LIN {X 0,Y 390.091,Z 385.39,A -85,B 0,C 180,E1 -11570.909,E2 -11570.909} C_VEL
LIN {X 0,Y 390.086,Z 385.387,A -85,B 0,C 180,E1 -11574.794,E2 -11574.794} C_VEL
LIN {X 0,Y 390.035,Z 385.403,A -85,B 0,C 180,E1 -11578.497,E2 -11578.497} C_VEL
LIN {X 0,Y 390.137,Z 385.63,A -85,B 0,C 180,E1 -11579.709,E2 -11579.709} C_VEL
LIN {X 0,Y 392.088,Z 395.547,A -85,B 0,C 180,E1 -11582.802,E2 -11582.802} C_VEL
LIN {X 0,Y 392.818,Z 399.954,A -85,B 0,C 180,E1 -11584.065,E2 -11584.065} C_VEL
LIN {X 0,Y 392.519,Z 405.952,A -85,B 0,C 180,E1 -11585.682,E2 -11585.682} C_VEL
LIN {X 0,Y 391.656,Z 416.045,A -85,B 0,C 180,E1 -11588.417,E2 -11588.417} C_VEL
LIN {X 0,Y 391.304,Z 419.949,A -85,B 0,C 180,E1 -11589.465,E2 -11589.465} C_VEL
LIN {X 0,Y 392.02,Z 423.777,A -85,B 0,C 180,E1 -11589.635,E2 -11589.635} C_VEL
LIN {X 0,Y 396.828,Z 450.131,A -85,B 0,C 180,E1 -11590.386,E2 -11590.386} C_VEL
LIN {X 0,Y 395.873,Z 524.91,A -85,B 0,C 180,E1 -11591.767,E2 -11591.767} C_VEL
LIN {X 0,Y 395.475,Z 534.822,A -85,B 0,C 180,E1 -11592.049,E2 -11592.049} C_VEL
LIN {X 0,Y 394.937,Z 544.807,A -85,B 0,C 180,E1 -11592.458,E2 -11592.458} C_VEL
LIN {X 0,Y 394.337,Z 555.164,A -85,B 0,C 180,E1 -11593.032,E2 -11593.032} C_VEL
LIN {X 0,Y 393.611,Z 564.308,A -85,B 0,C 180,E1 -11593.668,E2 -11593.668} C_VEL
LIN {X 0,Y 392.873,Z 573.31,A -85,B 0,C 180,E1 -11594.436,E2 -11594.436} C_VEL
LIN {X 0,Y 392.161,Z 582.039,A -85,B 0,C 180,E1 -11595.337,E2 -11595.337} C_VEL
LIN {X 0,Y 391.493,Z 589.792,A -85,B 0,C 180,E1 -11596.287,E2 -11596.287} C_VEL
LIN {X 0,Y 390.771,Z 598.261,A -85,B 0,C 180,E1 -11597.537,E2 -11597.537} C_VEL
LIN {X 0,Y 390.161,Z 604.25,A -85,B 0,C 180,E1 -11598.572,E2 -11598.572} C_VEL
LIN {X 0,Y 389.663,Z 610.562,A -85,B 0,C 180,E1 -11599.872,E2 -11599.872} C_VEL
LIN {X 0,Y 389.257,Z 615.836,A -85,B 0,C 180,E1 -11601.173,E2 -11601.173} C_VEL
LIN {X 0,Y 388.939,Z 620.93,A -85,B 0,C 180,E1 -11602.734,E2 -11602.734} C_VEL
LIN {X 0,Y 388.733,Z 624.78,A -85,B 0,C 180,E1 -11604.24,E2 -11604.24} C_VEL
LIN {X 0,Y 388.701,Z 627.827,A -85,B 0,C 180,E1 -11605.853,E2 -11605.853} C_VEL
LIN {X 0,Y 388.635,Z 629.324,A -85,B 0,C 180,E1 -11606.89,E2 -11606.89} C_VEL
LIN {X 0,Y 388.704,Z 630.847,A -85,B 0,C 180,E1 -11608.964,E2 -11608.964} C_VEL
LIN {X 0,Y 388.708,Z 631.126,A -85,B 0,C 180,E1 -11610,E2 -11610} C_VEL
LIN {X 0,Y 388.662,Z 630.251,A -85,B 0,C 180,E1 -11612.073,E2 -11612.073} C_VEL
LIN {X 0,Y 388.635,Z 629.324,A -85,B 0,C 180,E1 -11613.11,E2 -11613.11} C_VEL
LIN {X 0,Y 388.743,Z 625.981,A -85,B 0,C 180,E1 -11615.187,E2 -11615.187} C_VEL
LIN {X 0,Y 388.846,Z 622.355,A -85,B 0,C 180,E1 -11616.747,E2 -11616.747} C_VEL
LIN {X 0,Y 389.134,Z 617.624,A -85,B 0,C 180,E1 -11618.308,E2 -11618.308} C_VEL
LIN {X 0,Y 389.573,Z 611.652,A -85,B 0,C 180,E1 -11619.868,E2 -11619.868} C_VEL
LIN {X 0,Y 390.041,Z 605.559,A -85,B 0,C 180,E1 -11621.169,E2 -11621.169} C_VEL
LIN {X 0,Y 390.61,Z 599.818,A -85,B 0,C 180,E1 -11622.205,E2 -11622.205} C_VEL
LIN {X 0,Y 391.249,Z 593.161,A -85,B 0,C 180,E1 -11623.24,E2 -11623.24} C_VEL
LIN {X 0,Y 391.95,Z 585.084,A -85,B 0,C 180,E1 -11624.303,E2 -11624.303} C_VEL
LIN {X 0,Y 392.647,Z 576.194,A -85,B 0,C 180,E1 -11625.282,E2 -11625.282} C_VEL
LIN {X 0,Y 393.374,Z 567.482,A -85,B 0,C 180,E1 -11626.077,E2 -11626.077} C_VEL
LIN {X 0,Y 394.028,Z 559.091,A -85,B 0,C 180,E1 -11626.715,E2 -11626.715} C_VEL
LIN {X 0,Y 394.748,Z 548.583,A -85,B 0,C 180,E1 -11627.35,E2 -11627.35} C_VEL
LIN {X 0,Y 395.299,Z 538.249,A -85,B 0,C 180,E1 -11627.826,E2 -11627.826} C_VEL
LIN {X 0,Y 395.794,Z 527.528,A -85,B 0,C 180,E1 -11628.171,E2 -11628.171} C_VEL
LIN {X 0,Y 396.219,Z 504.75,A -85,B 0,C 180,E1 -11628.619,E2 -11628.619} C_VEL
LIN {X 0,Y 396.764,Z 449.751,A -85,B 0,C 180,E1 -11629.624,E2 -11629.624} C_VEL
LIN {X 0,Y 391.752,Z 422.313,A -85,B 0,C 180,E1 -11630.407,E2 -11630.407} C_VEL
LIN {X 0,Y 391.326,Z 419.943,A -85,B 0,C 180,E1 -11630.534,E2 -11630.534} C_VEL
LIN {X 0,Y 392.555,Z 406.144,A -85,B 0,C 180,E1 -11634.316,E2 -11634.316} C_VEL
LIN {X 0,Y 392.878,Z 400.185,A -85,B 0,C 180,E1 -11635.942,E2 -11635.942} C_VEL
LIN {X 0,Y 391.209,Z 390.975,A -85,B 0,C 180,E1 -11638.627,E2 -11638.627} C_VEL
LIN {X 0,Y 390.107,Z 385.497,A -85,B 0,C 180,E1 -11640.369,E2 -11640.369} C_VEL
LIN {X 0,Y 390.071,Z 385.399,A -85,B 0,C 180,E1 -11644.024,E2 -11644.024} C_VEL
LIN {X 0,Y 390.048,Z 385.397,A -85,B 0,C 180,E1 -11647.551,E2 -11647.551} C_VEL
LIN {X 0,Y 390.058,Z 385.376,A -85,B 0,C 180,E1 -11650.821,E2 -11650.821} C_VEL
LIN {X 0,Y 390.061,Z 385.4,A -85,B 0,C 180,E1 -11653.886,E2 -11653.886} C_VEL
LIN {X 0,Y 390.119,Z 385.387,A -85,B 0,C 180,E1 -11656.798,E2 -11656.798} C_VEL
LIN {X 0,Y 390.079,Z 385.389,A -85,B 0,C 180,E1 -11659.563,E2 -11659.563} C_VEL
LIN {X 0,Y 390.048,Z 385.398,A -85,B 0,C 180,E1 -11662.448,E2 -11662.448} C_VEL
LIN {X 0,Y 390.068,Z 385.382,A -85,B 0,C 180,E1 -11666.045,E2 -11666.045} C_VEL
LIN {X 0,Y 390.048,Z 385.397,A -85,B 0,C 180,E1 -11668.497,E2 -11668.497} C_VEL
LIN {X 0,Y 390.117,Z 385.375,A -85,B 0,C 180,E1 -11672.069,E2 -11672.069} C_VEL
LIN {X 0,Y 390.08,Z 385.387,A -85,B 0,C 180,E1 -11675.519,E2 -11675.519} C_VEL
LIN {X 0,Y 390.055,Z 385.39,A -85,B 0,C 180,E1 -11678.877,E2 -11678.877} C_VEL
LIN {X 0,Y 390.128,Z 385.368,A -85,B 0,C 180,E1 -11682.166,E2 -11682.166} C_VEL
LIN {X 0,Y 390.146,Z 385.383,A -85,B 0,C 180,E1 -11685.392,E2 -11685.392} C_VEL
LIN {X 0,Y 390.146,Z 385.372,A -85,B 0,C 180,E1 -11688.571,E2 -11688.571} C_VEL
LIN {X 0,Y 390.343,Z 385.344,A -85,B 0,C 180,E1 -11691.993,E2 -11691.993} C_VEL
LIN {X 0,Y 390.225,Z 385.373,A -85,B 0,C 180,E1 -11694.833,E2 -11694.833} C_VEL
LIN {X 0,Y 390.418,Z 385.342,A -85,B 0,C 180,E1 -11697.936,E2 -11697.936} C_VEL
LIN {X 0,Y 390.546,Z 385.309,A -85,B 0,C 180,E1 -11699.999,E2 -11699.999} C_VEL
LIN {X 0,Y 390.314,Z 385.356,A -85,B 0,C 180,E1 -11703.096,E2 -11703.096} C_VEL
LIN {X 0,Y 390.307,Z 385.361,A -85,B 0,C 180,E1 -11706.65,E2 -11706.65} C_VEL
LIN {X 0,Y 390.204,Z 385.358,A -85,B 0,C 180,E1 -11709.328,E2 -11709.328} C_VEL
LIN {X 0,Y 390.175,Z 385.374,A -85,B 0,C 180,E1 -11712.482,E2 -11712.482} C_VEL
LIN {X 0,Y 390.137,Z 385.387,A -85,B 0,C 180,E1 -11715.676,E2 -11715.676} C_VEL
LIN {X 0,Y 390.102,Z 385.371,A -85,B 0,C 180,E1 -11718.922,E2 -11718.922} C_VEL
LIN {X 0,Y 390.036,Z 385.397,A -85,B 0,C 180,E1 -11722.234,E2 -11722.234} C_VEL
LIN {X 0,Y 390.116,Z 385.38,A -85,B 0,C 180,E1 -11725.743,E2 -11725.743} C_VEL
LIN {X 0,Y 390.054,Z 385.388,A -85,B 0,C 180,E1 -11729.109,E2 -11729.109} C_VEL
LIN {X 0,Y 390.039,Z 385.397,A -85,B 0,C 180,E1 -11732.721,E2 -11732.721} C_VEL
LIN {X 0,Y 390.053,Z 385.393,A -85,B 0,C 180,E1 -11735.825,E2 -11735.825} C_VEL
LIN {X 0,Y 390.068,Z 385.394,A -85,B 0,C 180,E1 -11739.218,E2 -11739.218} C_VEL
LIN {X 0,Y 390.041,Z 385.396,A -85,B 0,C 180,E1 -11742.374,E2 -11742.374} C_VEL
LIN {X 0,Y 390.042,Z 385.388,A -85,B 0,C 180,E1 -11745.354,E2 -11745.354} C_VEL
LIN {X 0,Y 390.046,Z 385.361,A -85,B 0,C 180,E1 -11748.189,E2 -11748.189} C_VEL
LIN {X 0,Y 390.091,Z 385.388,A -85,B 0,C 180,E1 -11750.908,E2 -11750.908} C_VEL
LIN {X 0,Y 390.082,Z 385.374,A -85,B 0,C 180,E1 -11754.793,E2 -11754.793} C_VEL
LIN {X 0,Y 390.024,Z 385.402,A -85,B 0,C 180,E1 -11758.496,E2 -11758.496} C_VEL
LIN {X 0,Y 390.113,Z 385.389,A -85,B 0,C 180,E1 -11762.07,E2 -11762.07} C_VEL
LIN {X 0,Y 390.077,Z 385.397,A -85,B 0,C 180,E1 -11765.519,E2 -11765.519} C_VEL
LIN {X 0,Y 390.052,Z 385.401,A -85,B 0,C 180,E1 -11768.878,E2 -11768.878} C_VEL
LIN {X 0,Y 390.125,Z 385.391,A -85,B 0,C 180,E1 -11772.166,E2 -11772.166} C_VEL
LIN {X 0,Y 390.14,Z 385.39,A -85,B 0,C 180,E1 -11775.392,E2 -11775.392} C_VEL
LIN {X 0,Y 390.145,Z 385.389,A -85,B 0,C 180,E1 -11778.571,E2 -11778.571} C_VEL
LIN {X 0,Y 390.382,Z 385.657,A -85,B 0,C 180,E1 -11781.829,E2 -11781.829} C_VEL
LIN {X 0,Y 390.714,Z 386.9,A -85,B 0,C 180,E1 -11782.458,E2 -11782.458} C_VEL
LIN {X 0,Y 392.085,Z 389.234,A -85,B 0,C 180,E1 -11783.567,E2 -11783.567} C_VEL
LIN {X 0,Y 394.112,Z 390.919,A -85,B 0,C 180,E1 -11785.397,E2 -11785.397} C_VEL
LIN {X 0,Y 395.582,Z 391.492,A -85,B 0,C 180,E1 -11787.454,E2 -11787.454} C_VEL
LIN {X 0,Y 396.128,Z 391.931,A -85,B 0,C 180,E1 -11788.983,E2 -11788.983} C_VEL
LIN {X 0,Y 396.323,Z 391.849,A -85,B 0,C 180,E1 -11790,E2 -11790} C_VEL
LIN {X 0,Y 396.07,Z 391.804,A -85,B 0,C 180,E1 -11791.525,E2 -11791.525} C_VEL
LIN {X 0,Y 395.354,Z 391.371,A -85,B 0,C 180,E1 -11793.057,E2 -11793.057} C_VEL
LIN {X 0,Y 393.694,Z 390.658,A -85,B 0,C 180,E1 -11794.992,E2 -11794.992} C_VEL
LIN {X 0,Y 391.898,Z 389.022,A -85,B 0,C 180,E1 -11796.564,E2 -11796.564} C_VEL
LIN {X 0,Y 390.579,Z 386.504,A -85,B 0,C 180,E1 -11797.684,E2 -11797.684} C_VEL
LIN {X 0,Y 390.34,Z 385.593,A -85,B 0,C 180,E1 -11798.281,E2 -11798.281} C_VEL
LIN {X 0,Y 390.144,Z 385.389,A -85,B 0,C 180,E1 -11801.428,E2 -11801.428} C_VEL
LIN {X 0,Y 390.139,Z 385.39,A -85,B 0,C 180,E1 -11804.607,E2 -11804.607} C_VEL
LIN {X 0,Y 390.123,Z 385.391,A -85,B 0,C 180,E1 -11807.833,E2 -11807.833} C_VEL
LIN {X 0,Y 390.051,Z 385.402,A -85,B 0,C 180,E1 -11811.122,E2 -11811.122} C_VEL
LIN {X 0,Y 390.075,Z 385.397,A -85,B 0,C 180,E1 -11814.48,E2 -11814.48} C_VEL
LIN {X 0,Y 390.11,Z 385.387,A -85,B 0,C 180,E1 -11818.025,E2 -11818.025} C_VEL
LIN {X 0,Y 390.01,Z 385.395,A -85,B 0,C 180,E1 -11820.813,E2 -11820.813} C_VEL
LIN {X 0,Y 389.336,Z 385.488,A -85,B 0,C 180,E1 -11821.675,E2 -11821.675} C_VEL
LIN {X 0,Y 386.487,Z 385.833,A -85,B 0,C 180,E1 -11823.076,E2 -11823.076} C_VEL
LIN {X 0,Y 384.087,Z 386.121,A -85,B 0,C 180,E1 -11824.209,E2 -11824.209} C_VEL
LIN {X 0,Y 383.07,Z 386.246,A -85,B 0,C 180,E1 -11825.085,E2 -11825.085} C_VEL
LIN {X 0,Y 382.993,Z 386.257,A -85,B 0,C 180,E1 -11825.381,E2 -11825.381} C_VEL
LIN {X 0,Y 383.006,Z 386.277,A -85,B 0,C 180,E1 -11828.599,E2 -11828.599} C_VEL
LIN {X 0,Y 382.997,Z 386.241,A -85,B 0,C 180,E1 -11831.345,E2 -11831.345} C_VEL
LIN {X 0,Y 382.99,Z 386.262,A -85,B 0,C 180,E1 -11834.303,E2 -11834.303} C_VEL
LIN {X 0,Y 383.032,Z 386.27,A -85,B 0,C 180,E1 -11837.244,E2 -11837.244} C_VEL
LIN {X 0,Y 383.014,Z 386.267,A -85,B 0,C 180,E1 -11840.412,E2 -11840.412} C_VEL
LIN {X 0,Y 383.019,Z 386.271,A -85,B 0,C 180,E1 -11844.045,E2 -11844.045} C_VEL
LIN {X 0,Y 382.982,Z 386.275,A -85,B 0,C 180,E1 -11847.578,E2 -11847.578} C_VEL
LIN {X 0,Y 382.999,Z 386.275,A -85,B 0,C 180,E1 -11850.302,E2 -11850.302} C_VEL
LIN {X 0,Y 383.05,Z 386.253,A -85,B 0,C 180,E1 -11852.698,E2 -11852.698} C_VEL
LIN {X 0,Y 383.045,Z 386.269,A -85,B 0,C 180,E1 -11855.04,E2 -11855.04} C_VEL
LIN {X 0,Y 382.986,Z 386.271,A -85,B 0,C 180,E1 -11858.469,E2 -11858.469} C_VEL
LIN {X 0,Y 383.056,Z 386.25,A -85,B 0,C 180,E1 -11861.827,E2 -11861.827} C_VEL
LIN {X 0,Y 383.105,Z 386.262,A -85,B 0,C 180,E1 -11865.119,E2 -11865.119} C_VEL
LIN {X 0,Y 383.1,Z 386.247,A -85,B 0,C 180,E1 -11868.359,E2 -11868.359} C_VEL
LIN {X 0,Y 383.298,Z 386.225,A -85,B 0,C 180,E1 -11871.933,E2 -11871.933} C_VEL
LIN {X 0,Y 383.194,Z 386.252,A -85,B 0,C 180,E1 -11874.739,E2 -11874.739} C_VEL
LIN {X 0,Y 383.382,Z 386.215,A -85,B 0,C 180,E1 -11877.899,E2 -11877.899} C_VEL
LIN {X 0,Y 383.513,Z 386.184,A -85,B 0,C 180,E1 -11880.001,E2 -11880.001} C_VEL
LIN {X 0,Y 383.247,Z 386.242,A -85,B 0,C 180,E1 -11883.154,E2 -11883.154} C_VEL
LIN {X 0,Y 383.282,Z 386.236,A -85,B 0,C 180,E1 -11886.317,E2 -11886.317} C_VEL
LIN {X 0,Y 383.255,Z 386.219,A -85,B 0,C 180,E1 -11888.436,E2 -11888.436} C_VEL
LIN {X 0,Y 383.092,Z 386.252,A -85,B 0,C 180,E1 -11891.643,E2 -11891.643} C_VEL
LIN {X 0,Y 383.108,Z 386.258,A -85,B 0,C 180,E1 -11894.882,E2 -11894.882} C_VEL
LIN {X 0,Y 383.059,Z 386.246,A -85,B 0,C 180,E1 -11898.174,E2 -11898.174} C_VEL
LIN {X 0,Y 382.989,Z 386.271,A -85,B 0,C 180,E1 -11901.532,E2 -11901.532} C_VEL
LIN {X 0,Y 383.048,Z 386.259,A -85,B 0,C 180,E1 -11904.961,E2 -11904.961} C_VEL
LIN {X 0,Y 383.046,Z 386.264,A -85,B 0,C 180,E1 -11908.493,E2 -11908.493} C_VEL
LIN {X 0,Y 383.034,Z 386.267,A -85,B 0,C 180,E1 -11912.148,E2 -11912.148} C_VEL
LIN {X 0,Y 383.024,Z 386.27,A -85,B 0,C 180,E1 -11915.956,E2 -11915.956} C_VEL
LIN {X 0,Y 383.02,Z 386.266,A -85,B 0,C 180,E1 -11919.589,E2 -11919.589} C_VEL
LIN {X 0,Y 383.064,Z 386.266,A -85,B 0,C 180,E1 -11922.789,E2 -11922.789} C_VEL
LIN {X 0,Y 383.006,Z 386.276,A -85,B 0,C 180,E1 -11925.792,E2 -11925.792} C_VEL
LIN {X 0,Y 382.987,Z 386.259,A -85,B 0,C 180,E1 -11928.797,E2 -11928.797} C_VEL
LIN {X 0,Y 383.001,Z 386.278,A -85,B 0,C 180,E1 -11932.097,E2 -11932.097} C_VEL
LIN {X 0,Y 383.019,Z 386.273,A -85,B 0,C 180,E1 -11935.333,E2 -11935.333} C_VEL
LIN {X 0,Y 383.054,Z 386.367,A -85,B 0,C 180,E1 -11939.308,E2 -11939.308} C_VEL
LIN {X 0,Y 384.856,Z 395.359,A -85,B 0,C 180,E1 -11942.247,E2 -11942.247} C_VEL
LIN {X 0,Y 385.877,Z 401.628,A -85,B 0,C 180,E1 -11944.081,E2 -11944.081} C_VEL
LIN {X 0,Y 385.418,Z 408.77,A -85,B 0,C 180,E1 -11946.032,E2 -11946.032} C_VEL
LIN {X 0,Y 384.406,Z 419.746,A -85,B 0,C 180,E1 -11949.079,E2 -11949.079} C_VEL
LIN {X 0,Y 384.957,Z 422.907,A -85,B 0,C 180,E1 -11949.232,E2 -11949.232} C_VEL
LIN {X 0,Y 390.121,Z 450.943,A -85,B 0,C 180,E1 -11950.054,E2 -11950.054} C_VEL
LIN {X 0,Y 389.125,Z 524.715,A -85,B 0,C 180,E1 -11951.439,E2 -11951.439} C_VEL
LIN {X 0,Y 388.735,Z 534.627,A -85,B 0,C 180,E1 -11951.727,E2 -11951.727} C_VEL
LIN {X 0,Y 388.167,Z 544.612,A -85,B 0,C 180,E1 -11952.142,E2 -11952.142} C_VEL
LIN {X 0,Y 387.54,Z 554.969,A -85,B 0,C 180,E1 -11952.725,E2 -11952.725} C_VEL
LIN {X 0,Y 386.787,Z 564.113,A -85,B 0,C 180,E1 -11953.371,E2 -11953.371} C_VEL
LIN {X 0,Y 386.009,Z 573.115,A -85,B 0,C 180,E1 -11954.152,E2 -11954.152} C_VEL
LIN {X 0,Y 385.274,Z 581.844,A -85,B 0,C 180,E1 -11955.069,E2 -11955.069} C_VEL
LIN {X 0,Y 384.554,Z 589.767,A -85,B 0,C 180,E1 -11956.06,E2 -11956.06} C_VEL
LIN {X 0,Y 383.821,Z 598.065,A -85,B 0,C 180,E1 -11957.307,E2 -11957.307} C_VEL
LIN {X 0,Y 383.177,Z 604.054,A -85,B 0,C 180,E1 -11958.361,E2 -11958.361} C_VEL
LIN {X 0,Y 382.659,Z 610.367,A -85,B 0,C 180,E1 -11959.685,E2 -11959.685} C_VEL
LIN {X 0,Y 382.213,Z 615.64,A -85,B 0,C 180,E1 -11961.009,E2 -11961.009} C_VEL
LIN {X 0,Y 381.867,Z 620.734,A -85,B 0,C 180,E1 -11962.598,E2 -11962.598} C_VEL
LIN {X 0,Y 381.69,Z 624.065,A -85,B 0,C 180,E1 -11963.88,E2 -11963.88} C_VEL
LIN {X 0,Y 381.626,Z 627.632,A -85,B 0,C 180,E1 -11965.776,E2 -11965.776} C_VEL
LIN {X 0,Y 381.546,Z 629.129,A -85,B 0,C 180,E1 -11966.833,E2 -11966.833} C_VEL
LIN {X 0,Y 381.603,Z 630.652,A -85,B 0,C 180,E1 -11968.945,E2 -11968.945} C_VEL
LIN {X 0,Y 381.622,Z 630.932,A -85,B 0,C 180,E1 -11970,E2 -11970} C_VEL
LIN {X 0,Y 381.56,Z 630.056,A -85,B 0,C 180,E1 -11972.111,E2 -11972.111} C_VEL
LIN {X 0,Y 381.547,Z 629.129,A -85,B 0,C 180,E1 -11973.168,E2 -11973.168} C_VEL
LIN {X 0,Y 381.643,Z 625.785,A -85,B 0,C 180,E1 -11975.283,E2 -11975.283} C_VEL
LIN {X 0,Y 381.782,Z 622.16,A -85,B 0,C 180,E1 -11976.872,E2 -11976.872} C_VEL
LIN {X 0,Y 382.067,Z 617.428,A -85,B 0,C 180,E1 -11978.462,E2 -11978.462} C_VEL
LIN {X 0,Y 382.535,Z 611.456,A -85,B 0,C 180,E1 -11980.052,E2 -11980.052} C_VEL
LIN {X 0,Y 383.054,Z 605.363,A -85,B 0,C 180,E1 -11981.375,E2 -11981.375} C_VEL
LIN {X 0,Y 383.634,Z 599.622,A -85,B 0,C 180,E1 -11982.431,E2 -11982.431} C_VEL
LIN {X 0,Y 384.306,Z 592.965,A -85,B 0,C 180,E1 -11983.484,E2 -11983.484} C_VEL
LIN {X 0,Y 385.037,Z 584.888,A -85,B 0,C 180,E1 -11984.566,E2 -11984.566} C_VEL
LIN {X 0,Y 385.701,Z 577.049,A -85,B 0,C 180,E1 -11985.455,E2 -11985.455} C_VEL
LIN {X 0,Y 386.559,Z 567.287,A -85,B 0,C 180,E1 -11986.368,E2 -11986.368} C_VEL
LIN {X 0,Y 387.249,Z 558.896,A -85,B 0,C 180,E1 -11987.016,E2 -11987.016} C_VEL
LIN {X 0,Y 387.973,Z 548.388,A -85,B 0,C 180,E1 -11987.663,E2 -11987.663} C_VEL
LIN {X 0,Y 388.546,Z 538.054,A -85,B 0,C 180,E1 -11988.147,E2 -11988.147} C_VEL
LIN {X 0,Y 389.058,Z 527.333,A -85,B 0,C 180,E1 -11988.497,E2 -11988.497} C_VEL
LIN {X 0,Y 389.484,Z 504.554,A -85,B 0,C 180,E1 -11988.953,E2 -11988.953} C_VEL
LIN {X 0,Y 390.081,Z 450.645,A -85,B 0,C 180,E1 -11989.953,E2 -11989.953} C_VEL
LIN {X 0,Y 385.105,Z 423.546,A -85,B 0,C 180,E1 -11990.747,E2 -11990.747} C_VEL
LIN {X 0,Y 384.434,Z 420.018,A -85,B 0,C 180,E1 -11990.885,E2 -11990.885} C_VEL
LIN {X 0,Y 384.538,Z 417.771,A -85,B 0,C 180,E1 -11991.44,E2 -11991.44} C_VEL
LIN {X 0,Y 385.789,Z 404.956,A -85,B 0,C 180,E1 -11995.059,E2 -11995.059} C_VEL
LIN {X 0,Y 385.771,Z 400.514,A -85,B 0,C 180,E1 -11996.315,E2 -11996.315} C_VEL
LIN {X 0,Y 384.047,Z 391.334,A -85,B 0,C 180,E1 -11999.056,E2 -11999.056} C_VEL
LIN {X 0,Y 383.056,Z 386.368,A -85,B 0,C 180,E1 -12000.692,E2 -12000.692} C_VEL
LIN {X 0,Y 383.021,Z 386.273,A -85,B 0,C 180,E1 -12004.667,E2 -12004.667} C_VEL
LIN {X 0,Y 383.004,Z 386.278,A -85,B 0,C 180,E1 -12007.904,E2 -12007.904} C_VEL
LIN {X 0,Y 382.985,Z 386.259,A -85,B 0,C 180,E1 -12011.347,E2 -12011.347} C_VEL
LIN {X 0,Y 383.009,Z 386.274,A -85,B 0,C 180,E1 -12014.305,E2 -12014.305} C_VEL
LIN {X 0,Y 383.077,Z 386.265,A -85,B 0,C 180,E1 -12017.249,E2 -12017.249} C_VEL
LIN {X 0,Y 383.023,Z 386.265,A -85,B 0,C 180,E1 -12020.412,E2 -12020.412} C_VEL
LIN {X 0,Y 383.027,Z 386.269,A -85,B 0,C 180,E1 -12024.044,E2 -12024.044} C_VEL
LIN {X 0,Y 383.037,Z 386.267,A -85,B 0,C 180,E1 -12027.852,E2 -12027.852} C_VEL
LIN {X 0,Y 383.064,Z 386.258,A -85,B 0,C 180,E1 -12031.72,E2 -12031.72} C_VEL
LIN {X 0,Y 383.052,Z 386.259,A -85,B 0,C 180,E1 -12035.039,E2 -12035.039} C_VEL
LIN {X 0,Y 382.993,Z 386.271,A -85,B 0,C 180,E1 -12038.468,E2 -12038.468} C_VEL
LIN {X 0,Y 383.063,Z 386.245,A -85,B 0,C 180,E1 -12041.826,E2 -12041.826} C_VEL
LIN {X 0,Y 383.112,Z 386.257,A -85,B 0,C 180,E1 -12045.118,E2 -12045.118} C_VEL
LIN {X 0,Y 383.096,Z 386.251,A -85,B 0,C 180,E1 -12048.357,E2 -12048.357} C_VEL
LIN {X 0,Y 383.303,Z 386.218,A -85,B 0,C 180,E1 -12051.932,E2 -12051.932} C_VEL
LIN {X 0,Y 383.198,Z 386.249,A -85,B 0,C 180,E1 -12054.738,E2 -12054.738} C_VEL
LIN {X 0,Y 383.386,Z 386.218,A -85,B 0,C 180,E1 -12057.898,E2 -12057.898} C_VEL
LIN {X 0,Y 383.515,Z 386.184,A -85,B 0,C 180,E1 -12059.999,E2 -12059.999} C_VEL
LIN {X 0,Y 383.25,Z 386.236,A -85,B 0,C 180,E1 -12063.153,E2 -12063.153} C_VEL
LIN {X 0,Y 383.267,Z 386.237,A -85,B 0,C 180,E1 -12066.644,E2 -12066.644} C_VEL
LIN {X 0,Y 383.258,Z 386.228,A -85,B 0,C 180,E1 -12068.435,E2 -12068.435} C_VEL
LIN {X 0,Y 383.104,Z 386.247,A -85,B 0,C 180,E1 -12071.641,E2 -12071.641} C_VEL
LIN {X 0,Y 383.109,Z 386.261,A -85,B 0,C 180,E1 -12074.881,E2 -12074.881} C_VEL
LIN {X 0,Y 383.06,Z 386.25,A -85,B 0,C 180,E1 -12078.173,E2 -12078.173} C_VEL
LIN {X 0,Y 382.99,Z 386.271,A -85,B 0,C 180,E1 -12081.53,E2 -12081.53} C_VEL
LIN {X 0,Y 383.049,Z 386.269,A -85,B 0,C 180,E1 -12084.96,E2 -12084.96} C_VEL
LIN {X 0,Y 383.026,Z 386.261,A -85,B 0,C 180,E1 -12088.27,E2 -12088.27} C_VEL
LIN {X 0,Y 383.005,Z 386.273,A -85,B 0,C 180,E1 -12092.149,E2 -12092.149} C_VEL
LIN {X 0,Y 383.014,Z 386.258,A -85,B 0,C 180,E1 -12094.667,E2 -12094.667} C_VEL
LIN {X 0,Y 382.998,Z 386.277,A -85,B 0,C 180,E1 -12097.904,E2 -12097.904} C_VEL
LIN {X 0,Y 382.981,Z 386.27,A -85,B 0,C 180,E1 -12101.347,E2 -12101.347} C_VEL
LIN {X 0,Y 382.994,Z 386.274,A -85,B 0,C 180,E1 -12104.303,E2 -12104.303} C_VEL
LIN {X 0,Y 383.006,Z 386.24,A -85,B 0,C 180,E1 -12107.24,E2 -12107.24} C_VEL
LIN {X 0,Y 383.018,Z 386.266,A -85,B 0,C 180,E1 -12110.412,E2 -12110.412} C_VEL
LIN {X 0,Y 383.023,Z 386.262,A -85,B 0,C 180,E1 -12114.044,E2 -12114.044} C_VEL
LIN {X 0,Y 382.985,Z 386.278,A -85,B 0,C 180,E1 -12117.577,E2 -12117.577} C_VEL
LIN {X 0,Y 382.994,Z 386.262,A -85,B 0,C 180,E1 -12120.3,E2 -12120.3} C_VEL
LIN {X 0,Y 383.053,Z 386.271,A -85,B 0,C 180,E1 -12122.698,E2 -12122.698} C_VEL
LIN {X 0,Y 383.03,Z 386.274,A -85,B 0,C 180,E1 -12126.192,E2 -12126.192} C_VEL
LIN {X 0,Y 383.052,Z 386.272,A -85,B 0,C 180,E1 -12129.598,E2 -12129.598} C_VEL
LIN {X 0,Y 383.101,Z 386.267,A -85,B 0,C 180,E1 -12132.931,E2 -12132.931} C_VEL
LIN {X 0,Y 383.122,Z 386.263,A -85,B 0,C 180,E1 -12136.464,E2 -12136.464} C_VEL
LIN {X 0,Y 383.154,Z 386.531,A -85,B 0,C 180,E1 -12138.527,E2 -12138.527} C_VEL
LIN {X 0,Y 383.388,Z 387.531,A -85,B 0,C 180,E1 -12138.936,E2 -12138.936} C_VEL
LIN {X 0,Y 384.443,Z 389.598,A -85,B 0,C 180,E1 -12139.533,E2 -12139.533} C_VEL
LIN {X 0,Y 386.582,Z 391.495,A -85,B 0,C 180,E1 -12140.583,E2 -12140.583} C_VEL
LIN {X 0,Y 388.921,Z 392.828,A -85,B 0,C 180,E1 -12141.895,E2 -12141.895} C_VEL
LIN {X 0,Y 390.34,Z 395.395,A -85,B 0,C 180,E1 -12142.954,E2 -12142.954} C_VEL
LIN {X 0,Y 391.932,Z 397.07,A -85,B 0,C 180,E1 -12144.211,E2 -12144.211} C_VEL
LIN {X 0,Y 393.437,Z 398.03,A -85,B 0,C 180,E1 -12145.646,E2 -12145.646} C_VEL
LIN {X 0,Y 394.715,Z 398.539,A -85,B 0,C 180,E1 -12147.448,E2 -12147.448} C_VEL
LIN {X 0,Y 395.266,Z 398.978,A -85,B 0,C 180,E1 -12148.981,E2 -12148.981} C_VEL
LIN {X 0,Y 395.458,Z 398.896,A -85,B 0,C 180,E1 -12150,E2 -12150} C_VEL
LIN {X 0,Y 395.202,Z 398.853,A -85,B 0,C 180,E1 -12151.528,E2 -12151.528} C_VEL
LIN {X 0,Y 394.244,Z 398.355,A -85,B 0,C 180,E1 -12153.368,E2 -12153.368} C_VEL
LIN {X 0,Y 392.801,Z 397.722,A -85,B 0,C 180,E1 -12155.004,E2 -12155.004} C_VEL
LIN {X 0,Y 390.787,Z 395.983,A -85,B 0,C 180,E1 -12156.713,E2 -12156.713} C_VEL
LIN {X 0,Y 389.247,Z 393.415,A -85,B 0,C 180,E1 -12157.901,E2 -12157.901} C_VEL
LIN {X 0,Y 388.31,Z 392.289,A -85,B 0,C 180,E1 -12158.456,E2 -12158.456} C_VEL
LIN {X 0,Y 385.838,Z 391.008,A -85,B 0,C 180,E1 -12159.766,E2 -12159.766} C_VEL
LIN {X 0,Y 383.934,Z 388.794,A -85,B 0,C 180,E1 -12160.747,E2 -12160.747} C_VEL
LIN {X 0,Y 383.206,Z 386.796,A -85,B 0,C 180,E1 -12161.303,E2 -12161.303} C_VEL
LIN {X 0,Y 383.114,Z 386.297,A -85,B 0,C 180,E1 -12161.909,E2 -12161.909} C_VEL
LIN {X 0,Y 383.105,Z 386.266,A -85,B 0,C 180,E1 -12164.881,E2 -12164.881} C_VEL
LIN {X 0,Y 383.084,Z 386.268,A -85,B 0,C 180,E1 -12168.172,E2 -12168.172} C_VEL
LIN {X 0,Y 382.988,Z 386.28,A -85,B 0,C 180,E1 -12171.531,E2 -12171.531} C_VEL
LIN {X 0,Y 383.047,Z 386.273,A -85,B 0,C 180,E1 -12174.96,E2 -12174.96} C_VEL
LIN {X 0,Y 383.044,Z 386.259,A -85,B 0,C 180,E1 -12178.492,E2 -12178.492} C_VEL
LIN {X 0,Y 383.006,Z 386.277,A -85,B 0,C 180,E1 -12182.149,E2 -12182.149} C_VEL
LIN {X 0,Y 382.993,Z 386.257,A -85,B 0,C 180,E1 -12185.381,E2 -12185.381} C_VEL
LIN {X 0,Y 382.353,Z 386.347,A -85,B 0,C 180,E1 -12186.259,E2 -12186.259} C_VEL
LIN {X 0,Y 379.548,Z 386.709,A -85,B 0,C 180,E1 -12187.687,E2 -12187.687} C_VEL
LIN {X 0,Y 377.143,Z 387.008,A -85,B 0,C 180,E1 -12188.842,E2 -12188.842} C_VEL
LIN {X 0,Y 376.086,Z 387.129,A -85,B 0,C 180,E1 -12189.734,E2 -12189.734} C_VEL
LIN {X 0,Y 375.987,Z 387.134,A -85,B 0,C 180,E1 -12190.036,E2 -12190.036} C_VEL
LIN {X 0,Y 375.924,Z 387.139,A -85,B 0,C 180,E1 -12193.766,E2 -12193.766} C_VEL
LIN {X 0,Y 375.948,Z 387.156,A -85,B 0,C 180,E1 -12196.807,E2 -12196.807} C_VEL
LIN {X 0,Y 375.99,Z 387.139,A -85,B 0,C 180,E1 -12200.028,E2 -12200.028} C_VEL
LIN {X 0,Y 375.958,Z 387.149,A -85,B 0,C 180,E1 -12203.495,E2 -12203.495} C_VEL
LIN {X 0,Y 375.953,Z 387.138,A -85,B 0,C 180,E1 -12205.889,E2 -12205.889} C_VEL
LIN {X 0,Y 375.967,Z 387.15,A -85,B 0,C 180,E1 -12209.688,E2 -12209.688} C_VEL
LIN {X 0,Y 375.995,Z 387.132,A -85,B 0,C 180,E1 -12212.142,E2 -12212.142} C_VEL
LIN {X 0,Y 375.999,Z 387.141,A -85,B 0,C 180,E1 -12214.539,E2 -12214.539} C_VEL
LIN {X 0,Y 375.956,Z 387.152,A -85,B 0,C 180,E1 -12218.046,E2 -12218.046} C_VEL
LIN {X 0,Y 376.002,Z 387.127,A -85,B 0,C 180,E1 -12221.474,E2 -12221.474} C_VEL
LIN {X 0,Y 376.053,Z 387.142,A -85,B 0,C 180,E1 -12224.833,E2 -12224.833} C_VEL
LIN {X 0,Y 376.052,Z 387.128,A -85,B 0,C 180,E1 -12228.137,E2 -12228.137} C_VEL
LIN {X 0,Y 376.251,Z 387.102,A -85,B 0,C 180,E1 -12231.878,E2 -12231.878} C_VEL
LIN {X 0,Y 376.166,Z 387.129,A -85,B 0,C 180,E1 -12234.64,E2 -12234.64} C_VEL
LIN {X 0,Y 376.348,Z 387.091,A -85,B 0,C 180,E1 -12237.86,E2 -12237.86} C_VEL
LIN {X 0,Y 376.483,Z 387.059,A -85,B 0,C 180,E1 -12240.001,E2 -12240.001} C_VEL
LIN {X 0,Y 376.185,Z 387.121,A -85,B 0,C 180,E1 -12243.214,E2 -12243.214} C_VEL
LIN {X 0,Y 376.241,Z 387.112,A -85,B 0,C 180,E1 -12246.436,E2 -12246.436} C_VEL
LIN {X 0,Y 376.2,Z 387.096,A -85,B 0,C 180,E1 -12248.596,E2 -12248.596} C_VEL
LIN {X 0,Y 376.044,Z 387.131,A -85,B 0,C 180,E1 -12251.864,E2 -12251.864} C_VEL
LIN {X 0,Y 376.056,Z 387.135,A -85,B 0,C 180,E1 -12255.168,E2 -12255.168} C_VEL
LIN {X 0,Y 376.005,Z 387.123,A -85,B 0,C 180,E1 -12258.528,E2 -12258.528} C_VEL
LIN {X 0,Y 375.959,Z 387.15,A -85,B 0,C 180,E1 -12261.955,E2 -12261.955} C_VEL
LIN {X 0,Y 376.003,Z 387.137,A -85,B 0,C 180,E1 -12265.462,E2 -12265.462} C_VEL
LIN {X 0,Y 375.974,Z 387.147,A -85,B 0,C 180,E1 -12269.079,E2 -12269.079} C_VEL
LIN {X 0,Y 375.953,Z 387.143,A -85,B 0,C 180,E1 -12272.829,E2 -12272.829} C_VEL
LIN {X 0,Y 375.956,Z 387.145,A -85,B 0,C 180,E1 -12275.416,E2 -12275.416} C_VEL
LIN {X 0,Y 375.975,Z 387.148,A -85,B 0,C 180,E1 -12278.272,E2 -12278.272} C_VEL
LIN {X 0,Y 375.988,Z 387.148,A -85,B 0,C 180,E1 -12281.611,E2 -12281.611} C_VEL
LIN {X 0,Y 375.968,Z 387.149,A -85,B 0,C 180,E1 -12285.263,E2 -12285.263} C_VEL
LIN {X 0,Y 375.939,Z 387.134,A -85,B 0,C 180,E1 -12289.134,E2 -12289.134} C_VEL
LIN {X 0,Y 375.966,Z 387.156,A -85,B 0,C 180,E1 -12291.913,E2 -12291.913} C_VEL
LIN {X 0,Y 375.98,Z 387.149,A -85,B 0,C 180,E1 -12295.333,E2 -12295.333} C_VEL
LIN {X 0,Y 376.013,Z 387.276,A -85,B 0,C 180,E1 -12299.036,E2 -12299.036} C_VEL
LIN {X 0,Y 377.619,Z 395.319,A -85,B 0,C 180,E1 -12301.712,E2 -12301.712} C_VEL
LIN {X 0,Y 378.864,Z 402.487,A -85,B 0,C 180,E1 -12303.861,E2 -12303.861} C_VEL
LIN {X 0,Y 378.708,Z 407.155,A -85,B 0,C 180,E1 -12305.173,E2 -12305.173} C_VEL
LIN {X 0,Y 377.486,Z 419.566,A -85,B 0,C 180,E1 -12308.679,E2 -12308.679} C_VEL
LIN {X 0,Y 378.188,Z 423.444,A -85,B 0,C 180,E1 -12308.857,E2 -12308.857} C_VEL
LIN {X 0,Y 382.792,Z 447.926,A -85,B 0,C 180,E1 -12309.601,E2 -12309.601} C_VEL
LIN {X 0,Y 383.496,Z 452.152,A -85,B 0,C 180,E1 -12309.722,E2 -12309.722} C_VEL
LIN {X 0,Y 382.399,Z 524.52,A -85,B 0,C 180,E1 -12311.1,E2 -12311.1} C_VEL
LIN {X 0,Y 382.019,Z 534.433,A -85,B 0,C 180,E1 -12311.394,E2 -12311.394} C_VEL
LIN {X 0,Y 381.425,Z 544.417,A -85,B 0,C 180,E1 -12311.816,E2 -12311.816} C_VEL
LIN {X 0,Y 380.753,Z 554.773,A -85,B 0,C 180,E1 -12312.408,E2 -12312.408} C_VEL
LIN {X 0,Y 379.994,Z 563.918,A -85,B 0,C 180,E1 -12313.065,E2 -12313.065} C_VEL
LIN {X 0,Y 379.189,Z 572.92,A -85,B 0,C 180,E1 -12313.859,E2 -12313.859} C_VEL
LIN {X 0,Y 378.381,Z 581.648,A -85,B 0,C 180,E1 -12314.791,E2 -12314.791} C_VEL
LIN {X 0,Y 377.625,Z 589.742,A -85,B 0,C 180,E1 -12315.824,E2 -12315.824} C_VEL
LIN {X 0,Y 376.881,Z 597.87,A -85,B 0,C 180,E1 -12317.07,E2 -12317.07} C_VEL
LIN {X 0,Y 376.208,Z 603.858,A -85,B 0,C 180,E1 -12318.142,E2 -12318.142} C_VEL
LIN {X 0,Y 375.648,Z 610.171,A -85,B 0,C 180,E1 -12319.49,E2 -12319.49} C_VEL
LIN {X 0,Y 375.186,Z 615.445,A -85,B 0,C 180,E1 -12320.839,E2 -12320.839} C_VEL
LIN {X 0,Y 374.8,Z 620.538,A -85,B 0,C 180,E1 -12322.458,E2 -12322.458} C_VEL
LIN {X 0,Y 374.585,Z 624.21,A -85,B 0,C 180,E1 -12323.933,E2 -12323.933} C_VEL
LIN {X 0,Y 374.53,Z 627.436,A -85,B 0,C 180,E1 -12325.696,E2 -12325.696} C_VEL
LIN {X 0,Y 374.461,Z 628.934,A -85,B 0,C 180,E1 -12326.773,E2 -12326.773} C_VEL
LIN {X 0,Y 374.503,Z 630.457,A -85,B 0,C 180,E1 -12328.925,E2 -12328.925} C_VEL
LIN {X 0,Y 374.538,Z 630.737,A -85,B 0,C 180,E1 -12330,E2 -12330} C_VEL
LIN {X 0,Y 374.459,Z 629.861,A -85,B 0,C 180,E1 -12332.151,E2 -12332.151} C_VEL
LIN {X 0,Y 374.462,Z 628.934,A -85,B 0,C 180,E1 -12333.228,E2 -12333.228} C_VEL
LIN {X 0,Y 374.552,Z 625.589,A -85,B 0,C 180,E1 -12335.384,E2 -12335.384} C_VEL
LIN {X 0,Y 374.725,Z 621.964,A -85,B 0,C 180,E1 -12337.002,E2 -12337.002} C_VEL
LIN {X 0,Y 375.018,Z 617.232,A -85,B 0,C 180,E1 -12338.623,E2 -12338.623} C_VEL
LIN {X 0,Y 375.523,Z 611.26,A -85,B 0,C 180,E1 -12340.242,E2 -12340.242} C_VEL
LIN {X 0,Y 376.046,Z 605.166,A -85,B 0,C 180,E1 -12341.59,E2 -12341.59} C_VEL
LIN {X 0,Y 376.681,Z 599.426,A -85,B 0,C 180,E1 -12342.664,E2 -12342.664} C_VEL
LIN {X 0,Y 377.355,Z 592.769,A -85,B 0,C 180,E1 -12343.737,E2 -12343.737} C_VEL
LIN {X 0,Y 378.073,Z 585.505,A -85,B 0,C 180,E1 -12344.738,E2 -12344.738} C_VEL
LIN {X 0,Y 378.851,Z 576.853,A -85,B 0,C 180,E1 -12345.742,E2 -12345.742} C_VEL
LIN {X 0,Y 379.755,Z 567.092,A -85,B 0,C 180,E1 -12346.67,E2 -12346.67} C_VEL
LIN {X 0,Y 380.471,Z 558.701,A -85,B 0,C 180,E1 -12347.329,E2 -12347.329} C_VEL
LIN {X 0,Y 381.182,Z 548.192,A -85,B 0,C 180,E1 -12347.989,E2 -12347.989} C_VEL
LIN {X 0,Y 381.816,Z 537.859,A -85,B 0,C 180,E1 -12348.478,E2 -12348.478} C_VEL
LIN {X 0,Y 382.334,Z 527.138,A -85,B 0,C 180,E1 -12348.834,E2 -12348.834} C_VEL
LIN {X 0,Y 382.764,Z 504.359,A -85,B 0,C 180,E1 -12349.299,E2 -12349.299} C_VEL
LIN {X 0,Y 383.378,Z 451.227,A -85,B 0,C 180,E1 -12350.302,E2 -12350.302} C_VEL
LIN {X 0,Y 377.949,Z 422.096,A -85,B 0,C 180,E1 -12351.184,E2 -12351.184} C_VEL
LIN {X 0,Y 377.484,Z 419.576,A -85,B 0,C 180,E1 -12351.318,E2 -12351.318} C_VEL
LIN {X 0,Y 378.713,Z 407.26,A -85,B 0,C 180,E1 -12354.829,E2 -12354.829} C_VEL
LIN {X 0,Y 378.923,Z 402.758,A -85,B 0,C 180,E1 -12356.136,E2 -12356.136} C_VEL
LIN {X 0,Y 377.708,Z 395.599,A -85,B 0,C 180,E1 -12358.292,E2 -12358.292} C_VEL
LIN {X 0,Y 376.007,Z 387.257,A -85,B 0,C 180,E1 -12360.995,E2 -12360.995} C_VEL
LIN {X 0,Y 375.983,Z 387.15,A -85,B 0,C 180,E1 -12364.667,E2 -12364.667} C_VEL
LIN {X 0,Y 375.978,Z 387.152,A -85,B 0,C 180,E1 -12368.27,E2 -12368.27} C_VEL
LIN {X 0,Y 375.936,Z 387.139,A -85,B 0,C 180,E1 -12371.6,E2 -12371.6} C_VEL
LIN {X 0,Y 375.982,Z 387.147,A -85,B 0,C 180,E1 -12375.26,E2 -12375.26} C_VEL
LIN {X 0,Y 375.991,Z 387.147,A -85,B 0,C 180,E1 -12378.389,E2 -12378.389} C_VEL
LIN {X 0,Y 375.969,Z 387.151,A -85,B 0,C 180,E1 -12381.911,E2 -12381.911} C_VEL
LIN {X 0,Y 375.981,Z 387.14,A -85,B 0,C 180,E1 -12385.332,E2 -12385.332} C_VEL
LIN {X 0,Y 375.977,Z 387.15,A -85,B 0,C 180,E1 -12388.439,E2 -12388.439} C_VEL
LIN {X 0,Y 376.002,Z 387.132,A -85,B 0,C 180,E1 -12392.141,E2 -12392.141} C_VEL
LIN {X 0,Y 376.007,Z 387.137,A -85,B 0,C 180,E1 -12394.538,E2 -12394.538} C_VEL
LIN {X 0,Y 375.963,Z 387.15,A -85,B 0,C 180,E1 -12398.045,E2 -12398.045} C_VEL
LIN {X 0,Y 376.008,Z 387.122,A -85,B 0,C 180,E1 -12401.473,E2 -12401.473} C_VEL
LIN {X 0,Y 376.06,Z 387.135,A -85,B 0,C 180,E1 -12404.832,E2 -12404.832} C_VEL
LIN {X 0,Y 376.048,Z 387.13,A -85,B 0,C 180,E1 -12408.136,E2 -12408.136} C_VEL
LIN {X 0,Y 376.256,Z 387.094,A -85,B 0,C 180,E1 -12411.877,E2 -12411.877} C_VEL
LIN {X 0,Y 376.17,Z 387.124,A -85,B 0,C 180,E1 -12414.639,E2 -12414.639} C_VEL
LIN {X 0,Y 376.352,Z 387.094,A -85,B 0,C 180,E1 -12417.859,E2 -12417.859} C_VEL
LIN {X 0,Y 376.485,Z 387.059,A -85,B 0,C 180,E1 -12419.999,E2 -12419.999} C_VEL
LIN {X 0,Y 376.188,Z 387.116,A -85,B 0,C 180,E1 -12423.212,E2 -12423.212} C_VEL
LIN {X 0,Y 376.231,Z 387.113,A -85,B 0,C 180,E1 -12426.636,E2 -12426.636} C_VEL
LIN {X 0,Y 376.203,Z 387.107,A -85,B 0,C 180,E1 -12428.594,E2 -12428.594} C_VEL
LIN {X 0,Y 376.055,Z 387.128,A -85,B 0,C 180,E1 -12431.863,E2 -12431.863} C_VEL
LIN {X 0,Y 376.057,Z 387.142,A -85,B 0,C 180,E1 -12435.167,E2 -12435.167} C_VEL
LIN {X 0,Y 376.006,Z 387.127,A -85,B 0,C 180,E1 -12438.526,E2 -12438.526} C_VEL
LIN {X 0,Y 375.96,Z 387.152,A -85,B 0,C 180,E1 -12441.954,E2 -12441.954} C_VEL
LIN {X 0,Y 376.003,Z 387.141,A -85,B 0,C 180,E1 -12445.461,E2 -12445.461} C_VEL
LIN {X 0,Y 375.957,Z 387.143,A -85,B 0,C 180,E1 -12449.079,E2 -12449.079} C_VEL
LIN {X 0,Y 375.945,Z 387.153,A -85,B 0,C 180,E1 -12452.828,E2 -12452.828} C_VEL
LIN {X 0,Y 375.954,Z 387.142,A -85,B 0,C 180,E1 -12455.415,E2 -12455.415} C_VEL
LIN {X 0,Y 375.972,Z 387.151,A -85,B 0,C 180,E1 -12458.27,E2 -12458.27} C_VEL
LIN {X 0,Y 375.931,Z 387.15,A -85,B 0,C 180,E1 -12461.6,E2 -12461.6} C_VEL
LIN {X 0,Y 375.924,Z 387.147,A -85,B 0,C 180,E1 -12465.268,E2 -12465.268} C_VEL
LIN {X 0,Y 375.972,Z 387.121,A -85,B 0,C 180,E1 -12469.137,E2 -12469.137} C_VEL
LIN {X 0,Y 375.969,Z 387.153,A -85,B 0,C 180,E1 -12471.912,E2 -12471.912} C_VEL
LIN {X 0,Y 375.976,Z 387.127,A -85,B 0,C 180,E1 -12475.332,E2 -12475.332} C_VEL
LIN {X 0,Y 375.957,Z 387.154,A -85,B 0,C 180,E1 -12478.438,E2 -12478.438} C_VEL
LIN {X 0,Y 375.999,Z 387.146,A -85,B 0,C 180,E1 -12482.142,E2 -12482.142} C_VEL
LIN {X 0,Y 376.003,Z 387.15,A -85,B 0,C 180,E1 -12484.539,E2 -12484.539} C_VEL
LIN {X 0,Y 375.96,Z 387.156,A -85,B 0,C 180,E1 -12488.045,E2 -12488.045} C_VEL
LIN {X 0,Y 376.02,Z 387.149,A -85,B 0,C 180,E1 -12491.474,E2 -12491.474} C_VEL
LIN {X 0,Y 376.055,Z 387.144,A -85,B 0,C 180,E1 -12494.832,E2 -12494.832} C_VEL
LIN {X 0,Y 376.116,Z 387.431,A -85,B 0,C 180,E1 -12496.109,E2 -12496.109} C_VEL
LIN {X 0,Y 376.404,Z 388.517,A -85,B 0,C 180,E1 -12496.466,E2 -12496.466} C_VEL
LIN {X 0,Y 377.86,Z 391.022,A -85,B 0,C 180,E1 -12497.103,E2 -12497.103} C_VEL
LIN {X 0,Y 379.85,Z 392.579,A -85,B 0,C 180,E1 -12497.864,E2 -12497.864} C_VEL
LIN {X 0,Y 381.206,Z 393.425,A -85,B 0,C 180,E1 -12498.434,E2 -12498.434} C_VEL
LIN {X 0,Y 382.76,Z 396.024,A -85,B 0,C 180,E1 -12499.152,E2 -12499.152} C_VEL
LIN {X 0,Y 385.027,Z 398.223,A -85,B 0,C 180,E1 -12500.287,E2 -12500.287} C_VEL
LIN {X 0,Y 387.591,Z 399.678,A -85,B 0,C 180,E1 -12501.659,E2 -12501.659} C_VEL
LIN {X 0,Y 389.286,Z 402.436,A -85,B 0,C 180,E1 -12502.842,E2 -12502.842} C_VEL
LIN {X 0,Y 391.041,Z 404.135,A -85,B 0,C 180,E1 -12504.198,E2 -12504.198} C_VEL
LIN {X 0,Y 392.756,Z 405.215,A -85,B 0,C 180,E1 -12505.895,E2 -12505.895} C_VEL
LIN {X 0,Y 393.915,Z 405.599,A -85,B 0,C 180,E1 -12507.579,E2 -12507.579} C_VEL
LIN {X 0,Y 394.407,Z 406.003,A -85,B 0,C 180,E1 -12508.979,E2 -12508.979} C_VEL
LIN {X 0,Y 394.593,Z 405.943,A -85,B 0,C 180,E1 -12510,E2 -12510} C_VEL
LIN {X 0,Y 394.096,Z 405.716,A -85,B 0,C 180,E1 -12512.044,E2 -12512.044} C_VEL
LIN {X 0,Y 393.066,Z 405.32,A -85,B 0,C 180,E1 -12513.724,E2 -12513.724} C_VEL
LIN {X 0,Y 391.761,Z 404.661,A -85,B 0,C 180,E1 -12515.146,E2 -12515.146} C_VEL
LIN {X 0,Y 389.867,Z 403.121,A -85,B 0,C 180,E1 -12516.729,E2 -12516.729} C_VEL
LIN {X 0,Y 388.033,Z 400.487,A -85,B 0,C 180,E1 -12518.061,E2 -12518.061} C_VEL
LIN {X 0,Y 387.37,Z 399.381,A -85,B 0,C 180,E1 -12518.476,E2 -12518.476} C_VEL
LIN {X 0,Y 384.676,Z 397.976,A -85,B 0,C 180,E1 -12519.88,E2 -12519.88} C_VEL
LIN {X 0,Y 382.363,Z 395.516,A -85,B 0,C 180,E1 -12521.027,E2 -12521.027} C_VEL
LIN {X 0,Y 380.869,Z 393.117,A -85,B 0,C 180,E1 -12521.711,E2 -12521.711} C_VEL
LIN {X 0,Y 378.467,Z 391.617,A -85,B 0,C 180,E1 -12522.67,E2 -12522.67} C_VEL
LIN {X 0,Y 376.702,Z 389.286,A -85,B 0,C 180,E1 -12523.377,E2 -12523.377} C_VEL
LIN {X 0,Y 376.2,Z 387.748,A -85,B 0,C 180,E1 -12523.729,E2 -12523.729} C_VEL
LIN {X 0,Y 376.063,Z 387.166,A -85,B 0,C 180,E1 -12524.336,E2 -12524.336} C_VEL
LIN {X 0,Y 376.039,Z 387.146,A -85,B 0,C 180,E1 -12527.607,E2 -12527.607} C_VEL
LIN {X 0,Y 375.973,Z 387.155,A -85,B 0,C 180,E1 -12530.832,E2 -12530.832} C_VEL
LIN {X 0,Y 375.988,Z 387.152,A -85,B 0,C 180,E1 -12534.281,E2 -12534.281} C_VEL
LIN {X 0,Y 376.014,Z 387.15,A -85,B 0,C 180,E1 -12536.652,E2 -12536.652} C_VEL
LIN {X 0,Y 375.971,Z 387.135,A -85,B 0,C 180,E1 -12539.078,E2 -12539.078} C_VEL
LIN {X 0,Y 375.944,Z 387.148,A -85,B 0,C 180,E1 -12542.828,E2 -12542.828} C_VEL
LIN {X 0,Y 375.952,Z 387.135,A -85,B 0,C 180,E1 -12545.415,E2 -12545.415} C_VEL
LIN {X 0,Y 375.976,Z 387.153,A -85,B 0,C 180,E1 -12548.272,E2 -12548.272} C_VEL
LIN {X 0,Y 375.987,Z 387.134,A -85,B 0,C 180,E1 -12550.036,E2 -12550.036} C_VEL
LIN {X 0,Y 375.269,Z 387.207,A -85,B 0,C 180,E1 -12550.93,E2 -12550.93} C_VEL
LIN {X 0,Y 372.358,Z 387.563,A -85,B 0,C 180,E1 -12552.381,E2 -12552.381} C_VEL
LIN {X 0,Y 369.946,Z 387.877,A -85,B 0,C 180,E1 -12553.555,E2 -12553.555} C_VEL
LIN {X 0,Y 368.955,Z 388.011,A -85,B 0,C 180,E1 -12554.464,E2 -12554.464} C_VEL
LIN {X 0,Y 368.896,Z 388.022,A -85,B 0,C 180,E1 -12554.772,E2 -12554.772} C_VEL
LIN {X 0,Y 368.903,Z 388.028,A -85,B 0,C 180,E1 -12558.181,E2 -12558.181} C_VEL
LIN {X 0,Y 368.905,Z 388.031,A -85,B 0,C 180,E1 -12561.359,E2 -12561.359} C_VEL
LIN {X 0,Y 368.93,Z 388.012,A -85,B 0,C 180,E1 -12565.147,E2 -12565.147} C_VEL
LIN {X 0,Y 368.922,Z 388.03,A -85,B 0,C 180,E1 -12569.047,E2 -12569.047} C_VEL
LIN {X 0,Y 368.981,Z 388.009,A -85,B 0,C 180,E1 -12571.565,E2 -12571.565} C_VEL
LIN {X 0,Y 368.95,Z 388.024,A -85,B 0,C 180,E1 -12575.225,E2 -12575.225} C_VEL
LIN {X 0,Y 368.931,Z 388.016,A -85,B 0,C 180,E1 -12578.974,E2 -12578.974} C_VEL
LIN {X 0,Y 368.984,Z 388.005,A -85,B 0,C 180,E1 -12582.258,E2 -12582.258} C_VEL
LIN {X 0,Y 369.031,Z 388.018,A -85,B 0,C 180,E1 -12586.228,E2 -12586.228} C_VEL
LIN {X 0,Y 369.063,Z 387.985,A -85,B 0,C 180,E1 -12590.132,E2 -12590.132} C_VEL
LIN {X 0,Y 369.182,Z 387.987,A -85,B 0,C 180,E1 -12592.343,E2 -12592.343} C_VEL
LIN {X 0,Y 369.139,Z 388.005,A -85,B 0,C 180,E1 -12594.538,E2 -12594.538} C_VEL
LIN {X 0,Y 369.313,Z 387.967,A -85,B 0,C 180,E1 -12597.819,E2 -12597.819} C_VEL
LIN {X 0,Y 369.452,Z 387.934,A -85,B 0,C 180,E1 -12600.001,E2 -12600.001} C_VEL
LIN {X 0,Y 369.314,Z 387.971,A -85,B 0,C 180,E1 -12602.182,E2 -12602.182} C_VEL
LIN {X 0,Y 369.203,Z 387.987,A -85,B 0,C 180,E1 -12606.559,E2 -12606.559} C_VEL
LIN {X 0,Y 369.132,Z 387.974,A -85,B 0,C 180,E1 -12608.762,E2 -12608.762} C_VEL
LIN {X 0,Y 369,Z 388.01,A -85,B 0,C 180,E1 -12612.094,E2 -12612.094} C_VEL
LIN {X 0,Y 368.996,Z 388.015,A -85,B 0,C 180,E1 -12615.465,E2 -12615.465} C_VEL
LIN {X 0,Y 368.954,Z 388.001,A -85,B 0,C 180,E1 -12618.895,E2 -12618.895} C_VEL
LIN {X 0,Y 368.928,Z 388.03,A -85,B 0,C 180,E1 -12622.396,E2 -12622.396} C_VEL
LIN {X 0,Y 368.996,Z 388.003,A -85,B 0,C 180,E1 -12625.981,E2 -12625.981} C_VEL
LIN {X 0,Y 368.964,Z 388.021,A -85,B 0,C 180,E1 -12628.814,E2 -12628.814} C_VEL
LIN {X 0,Y 368.907,Z 388.025,A -85,B 0,C 180,E1 -12632.238,E2 -12632.238} C_VEL
LIN {X 0,Y 368.927,Z 388.02,A -85,B 0,C 180,E1 -12635.002,E2 -12635.002} C_VEL
LIN {X 0,Y 368.911,Z 388.025,A -85,B 0,C 180,E1 -12638.642,E2 -12638.642} C_VEL
LIN {X 0,Y 368.95,Z 388.029,A -85,B 0,C 180,E1 -12642.023,E2 -12642.023} C_VEL
LIN {X 0,Y 368.923,Z 388.027,A -85,B 0,C 180,E1 -12645.184,E2 -12645.184} C_VEL
LIN {X 0,Y 368.881,Z 388.02,A -85,B 0,C 180,E1 -12648.178,E2 -12648.178} C_VEL
LIN {X 0,Y 368.91,Z 388.03,A -85,B 0,C 180,E1 -12651.36,E2 -12651.36} C_VEL
LIN {X 0,Y 368.937,Z 388.024,A -85,B 0,C 180,E1 -12655.147,E2 -12655.147} C_VEL
LIN {X 0,Y 368.951,Z 388.212,A -85,B 0,C 180,E1 -12658.731,E2 -12658.731} C_VEL
LIN {X 0,Y 370.453,Z 395.676,A -85,B 0,C 180,E1 -12661.275,E2 -12661.275} C_VEL
LIN {X 0,Y 371.976,Z 404.39,A -85,B 0,C 180,E1 -12663.943,E2 -12663.943} C_VEL
LIN {X 0,Y 371.393,Z 411.553,A -85,B 0,C 180,E1 -12665.993,E2 -12665.993} C_VEL
LIN {X 0,Y 370.617,Z 419.437,A -85,B 0,C 180,E1 -12668.276,E2 -12668.276} C_VEL
LIN {X 0,Y 371.687,Z 425.119,A -85,B 0,C 180,E1 -12668.507,E2 -12668.507} C_VEL
LIN {X 0,Y 376.221,Z 449.345,A -85,B 0,C 180,E1 -12669.26,E2 -12669.26} C_VEL
LIN {X 0,Y 376.807,Z 454.758,A -85,B 0,C 180,E1 -12669.402,E2 -12669.402} C_VEL
LIN {X 0,Y 375.69,Z 524.325,A -85,B 0,C 180,E1 -12670.749,E2 -12670.749} C_VEL
LIN {X 0,Y 375.309,Z 534.238,A -85,B 0,C 180,E1 -12671.049,E2 -12671.049} C_VEL
LIN {X 0,Y 374.687,Z 544.222,A -85,B 0,C 180,E1 -12671.477,E2 -12671.477} C_VEL
LIN {X 0,Y 373.986,Z 554.578,A -85,B 0,C 180,E1 -12672.079,E2 -12672.079} C_VEL
LIN {X 0,Y 373.212,Z 563.723,A -85,B 0,C 180,E1 -12672.748,E2 -12672.748} C_VEL
LIN {X 0,Y 372.364,Z 572.724,A -85,B 0,C 180,E1 -12673.555,E2 -12673.555} C_VEL
LIN {X 0,Y 371.509,Z 581.452,A -85,B 0,C 180,E1 -12674.502,E2 -12674.502} C_VEL
LIN {X 0,Y 370.777,Z 589.077,A -85,B 0,C 180,E1 -12675.486,E2 -12675.486} C_VEL
LIN {X 0,Y 369.932,Z 597.674,A -85,B 0,C 180,E1 -12676.822,E2 -12676.822} C_VEL
LIN {X 0,Y 369.251,Z 603.663,A -85,B 0,C 180,E1 -12677.915,E2 -12677.915} C_VEL
LIN {X 0,Y 368.609,Z 609.974,A -85,B 0,C 180,E1 -12679.287,E2 -12679.287} C_VEL
LIN {X 0,Y 368.134,Z 615.248,A -85,B 0,C 180,E1 -12680.662,E2 -12680.662} C_VEL
LIN {X 0,Y 367.723,Z 620.342,A -85,B 0,C 180,E1 -12682.312,E2 -12682.312} C_VEL
LIN {X 0,Y 367.506,Z 624.279,A -85,B 0,C 180,E1 -12683.949,E2 -12683.949} C_VEL
LIN {X 0,Y 367.438,Z 627.241,A -85,B 0,C 180,E1 -12685.613,E2 -12685.613} C_VEL
LIN {X 0,Y 367.379,Z 628.739,A -85,B 0,C 180,E1 -12686.71,E2 -12686.71} C_VEL
LIN {X 0,Y 367.403,Z 630.262,A -85,B 0,C 180,E1 -12688.904,E2 -12688.904} C_VEL
LIN {X 0,Y 367.44,Z 630.542,A -85,B 0,C 180,E1 -12690,E2 -12690} C_VEL
LIN {X 0,Y 367.36,Z 629.666,A -85,B 0,C 180,E1 -12692.193,E2 -12692.193} C_VEL
LIN {X 0,Y 367.379,Z 628.739,A -85,B 0,C 180,E1 -12693.29,E2 -12693.29} C_VEL
LIN {X 0,Y 367.464,Z 625.394,A -85,B 0,C 180,E1 -12695.488,E2 -12695.488} C_VEL
LIN {X 0,Y 367.662,Z 621.769,A -85,B 0,C 180,E1 -12697.138,E2 -12697.138} C_VEL
LIN {X 0,Y 367.988,Z 617.037,A -85,B 0,C 180,E1 -12698.789,E2 -12698.789} C_VEL
LIN {X 0,Y 368.519,Z 611.065,A -85,B 0,C 180,E1 -12700.438,E2 -12700.438} C_VEL
LIN {X 0,Y 369.064,Z 604.971,A -85,B 0,C 180,E1 -12701.813,E2 -12701.813} C_VEL
LIN {X 0,Y 369.735,Z 599.23,A -85,B 0,C 180,E1 -12702.906,E2 -12702.906} C_VEL
LIN {X 0,Y 370.41,Z 592.572,A -85,B 0,C 180,E1 -12704,E2 -12704} C_VEL
LIN {X 0,Y 371.191,Z 584.93,A -85,B 0,C 180,E1 -12705.066,E2 -12705.066} C_VEL
LIN {X 0,Y 371.999,Z 576.658,A -85,B 0,C 180,E1 -12706.04,E2 -12706.04} C_VEL
LIN {X 0,Y 372.948,Z 566.896,A -85,B 0,C 180,E1 -12706.983,E2 -12706.983} C_VEL
LIN {X 0,Y 373.698,Z 558.506,A -85,B 0,C 180,E1 -12707.653,E2 -12707.653} C_VEL
LIN {X 0,Y 374.424,Z 547.997,A -85,B 0,C 180,E1 -12708.325,E2 -12708.325} C_VEL
LIN {X 0,Y 375.101,Z 537.664,A -85,B 0,C 180,E1 -12708.821,E2 -12708.821} C_VEL
LIN {X 0,Y 375.624,Z 526.943,A -85,B 0,C 180,E1 -12709.184,E2 -12709.184} C_VEL
LIN {X 0,Y 376.053,Z 504.164,A -85,B 0,C 180,E1 -12709.658,E2 -12709.658} C_VEL
LIN {X 0,Y 376.698,Z 451.945,A -85,B 0,C 180,E1 -12710.661,E2 -12710.661} C_VEL
LIN {X 0,Y 371.498,Z 424.01,A -85,B 0,C 180,E1 -12711.527,E2 -12711.527} C_VEL
LIN {X 0,Y 370.577,Z 419.456,A -85,B 0,C 180,E1 -12711.722,E2 -12711.722} C_VEL
LIN {X 0,Y 371.832,Z 407.432,A -85,B 0,C 180,E1 -12715.213,E2 -12715.213} C_VEL
LIN {X 0,Y 371.922,Z 403.569,A -85,B 0,C 180,E1 -12716.364,E2 -12716.364} C_VEL
LIN {X 0,Y 370.023,Z 393.216,A -85,B 0,C 180,E1 -12719.592,E2 -12719.592} C_VEL
LIN {X 0,Y 368.94,Z 388.12,A -85,B 0,C 180,E1 -12721.35,E2 -12721.35} C_VEL
LIN {X 0,Y 368.932,Z 388.023,A -85,B 0,C 180,E1 -12725.001,E2 -12725.001} C_VEL
LIN {X 0,Y 368.912,Z 388.03,A -85,B 0,C 180,E1 -12728.64,E2 -12728.64} C_VEL
LIN {X 0,Y 368.883,Z 388.021,A -85,B 0,C 180,E1 -12732.009,E2 -12732.009} C_VEL
LIN {X 0,Y 368.957,Z 388.022,A -85,B 0,C 180,E1 -12735.187,E2 -12735.187} C_VEL
LIN {X 0,Y 368.947,Z 388.027,A -85,B 0,C 180,E1 -12738.186,E2 -12738.186} C_VEL
LIN {X 0,Y 368.914,Z 388.024,A -85,B 0,C 180,E1 -12741.358,E2 -12741.358} C_VEL
LIN {X 0,Y 368.938,Z 388.018,A -85,B 0,C 180,E1 -12745.146,E2 -12745.146} C_VEL
LIN {X 0,Y 368.93,Z 388.027,A -85,B 0,C 180,E1 -12749.046,E2 -12749.046} C_VEL
LIN {X 0,Y 368.987,Z 388.013,A -85,B 0,C 180,E1 -12751.564,E2 -12751.564} C_VEL
LIN {X 0,Y 368.958,Z 388.015,A -85,B 0,C 180,E1 -12755.224,E2 -12755.224} C_VEL
LIN {X 0,Y 368.937,Z 388.021,A -85,B 0,C 180,E1 -12758.973,E2 -12758.973} C_VEL
LIN {X 0,Y 368.99,Z 387.999,A -85,B 0,C 180,E1 -12762.257,E2 -12762.257} C_VEL
LIN {X 0,Y 369.036,Z 388.013,A -85,B 0,C 180,E1 -12766.227,E2 -12766.227} C_VEL
LIN {X 0,Y 369.066,Z 387.979,A -85,B 0,C 180,E1 -12770.131,E2 -12770.131} C_VEL
LIN {X 0,Y 369.187,Z 387.983,A -85,B 0,C 180,E1 -12772.342,E2 -12772.342} C_VEL
LIN {X 0,Y 369.143,Z 388,A -85,B 0,C 180,E1 -12774.537,E2 -12774.537} C_VEL
LIN {X 0,Y 369.317,Z 387.97,A -85,B 0,C 180,E1 -12777.818,E2 -12777.818} C_VEL
LIN {X 0,Y 369.454,Z 387.934,A -85,B 0,C 180,E1 -12779.999,E2 -12779.999} C_VEL
LIN {X 0,Y 369.317,Z 387.967,A -85,B 0,C 180,E1 -12782.181,E2 -12782.181} C_VEL
LIN {X 0,Y 369.201,Z 387.99,A -85,B 0,C 180,E1 -12786.624,E2 -12786.624} C_VEL
LIN {X 0,Y 369.136,Z 387.987,A -85,B 0,C 180,E1 -12788.76,E2 -12788.76} C_VEL
LIN {X 0,Y 369.01,Z 388.009,A -85,B 0,C 180,E1 -12792.092,E2 -12792.092} C_VEL
LIN {X 0,Y 368.996,Z 388.023,A -85,B 0,C 180,E1 -12795.464,E2 -12795.464} C_VEL
LIN {X 0,Y 368.955,Z 388.003,A -85,B 0,C 180,E1 -12798.894,E2 -12798.894} C_VEL
LIN {X 0,Y 368.929,Z 388.026,A -85,B 0,C 180,E1 -12802.395,E2 -12802.395} C_VEL
LIN {X 0,Y 368.997,Z 388.008,A -85,B 0,C 180,E1 -12805.98,E2 -12805.98} C_VEL
LIN {X 0,Y 368.911,Z 388.029,A -85,B 0,C 180,E1 -12809.69,E2 -12809.69} C_VEL
LIN {X 0,Y 368.893,Z 388.029,A -85,B 0,C 180,E1 -12813.043,E2 -12813.043} C_VEL
LIN {X 0,Y 368.914,Z 388.027,A -85,B 0,C 180,E1 -12816.196,E2 -12816.196} C_VEL
LIN {X 0,Y 368.901,Z 388.034,A -85,B 0,C 180,E1 -12818.952,E2 -12818.952} C_VEL
LIN {X 0,Y 368.878,Z 388.033,A -85,B 0,C 180,E1 -12822.009,E2 -12822.009} C_VEL
LIN {X 0,Y 368.882,Z 388.025,A -85,B 0,C 180,E1 -12825.176,E2 -12825.176} C_VEL
LIN {X 0,Y 368.89,Z 387.993,A -85,B 0,C 180,E1 -12828.179,E2 -12828.179} C_VEL
LIN {X 0,Y 368.913,Z 388.031,A -85,B 0,C 180,E1 -12831.358,E2 -12831.358} C_VEL
LIN {X 0,Y 368.933,Z 388.004,A -85,B 0,C 180,E1 -12835.146,E2 -12835.146} C_VEL
LIN {X 0,Y 368.925,Z 388.026,A -85,B 0,C 180,E1 -12839.046,E2 -12839.046} C_VEL
LIN {X 0,Y 368.983,Z 388.01,A -85,B 0,C 180,E1 -12841.564,E2 -12841.564} C_VEL
LIN {X 0,Y 368.954,Z 388.029,A -85,B 0,C 180,E1 -12845.224,E2 -12845.224} C_VEL
LIN {X 0,Y 368.934,Z 388.031,A -85,B 0,C 180,E1 -12848.973,E2 -12848.973} C_VEL
LIN {X 0,Y 368.987,Z 388.025,A -85,B 0,C 180,E1 -12852.257,E2 -12852.257} C_VEL
LIN {X 0,Y 369.013,Z 388.291,A -85,B 0,C 180,E1 -12854.04,E2 -12854.04} C_VEL
LIN {X 0,Y 369.278,Z 389.281,A -85,B 0,C 180,E1 -12854.353,E2 -12854.353} C_VEL
LIN {X 0,Y 370.507,Z 391.576,A -85,B 0,C 180,E1 -12854.81,E2 -12854.81} C_VEL
LIN {X 0,Y 372.884,Z 393.484,A -85,B 0,C 180,E1 -12855.608,E2 -12855.608} C_VEL
LIN {X 0,Y 373.97,Z 394.369,A -85,B 0,C 180,E1 -12855.962,E2 -12855.962} C_VEL
LIN {X 0,Y 375.971,Z 397.483,A -85,B 0,C 180,E1 -12856.76,E2 -12856.76} C_VEL
LIN {X 0,Y 378.432,Z 399.425,A -85,B 0,C 180,E1 -12857.668,E2 -12857.668} C_VEL
LIN {X 0,Y 379.535,Z 400.186,A -85,B 0,C 180,E1 -12858.131,E2 -12858.131} C_VEL
LIN {X 0,Y 381.399,Z 402.935,A -85,B 0,C 180,E1 -12858.978,E2 -12858.978} C_VEL
LIN {X 0,Y 383.705,Z 405.063,A -85,B 0,C 180,E1 -12860.095,E2 -12860.095} C_VEL
LIN {X 0,Y 386.285,Z 406.572,A -85,B 0,C 180,E1 -12861.433,E2 -12861.433} C_VEL
LIN {X 0,Y 388.223,Z 409.439,A -85,B 0,C 180,E1 -12862.72,E2 -12862.72} C_VEL
LIN {X 0,Y 390.151,Z 411.179,A -85,B 0,C 180,E1 -12864.184,E2 -12864.184} C_VEL
LIN {X 0,Y 391.884,Z 412.239,A -85,B 0,C 180,E1 -12865.886,E2 -12865.886} C_VEL
LIN {X 0,Y 392.994,Z 412.614,A -85,B 0,C 180,E1 -12867.456,E2 -12867.456} C_VEL
LIN {X 0,Y 393.545,Z 413.05,A -85,B 0,C 180,E1 -12868.976,E2 -12868.976} C_VEL
LIN {X 0,Y 393.727,Z 412.99,A -85,B 0,C 180,E1 -12870,E2 -12870} C_VEL
LIN {X 0,Y 393.467,Z 412.924,A -85,B 0,C 180,E1 -12871.535,E2 -12871.535} C_VEL
LIN {X 0,Y 392.738,Z 412.499,A -85,B 0,C 180,E1 -12873.077,E2 -12873.077} C_VEL
LIN {X 0,Y 391.175,Z 411.894,A -85,B 0,C 180,E1 -12874.895,E2 -12874.895} C_VEL
LIN {X 0,Y 389.129,Z 410.384,A -85,B 0,C 180,E1 -12876.619,E2 -12876.619} C_VEL
LIN {X 0,Y 387.297,Z 408.114,A -85,B 0,C 180,E1 -12877.941,E2 -12877.941} C_VEL
LIN {X 0,Y 385.95,Z 406.185,A -85,B 0,C 180,E1 -12878.772,E2 -12878.772} C_VEL
LIN {X 0,Y 383.231,Z 404.738,A -85,B 0,C 180,E1 -12880.134,E2 -12880.134} C_VEL
LIN {X 0,Y 380.894,Z 402.373,A -85,B 0,C 180,E1 -12881.238,E2 -12881.238} C_VEL
LIN {X 0,Y 379.161,Z 399.793,A -85,B 0,C 180,E1 -12882.036,E2 -12882.036} C_VEL
LIN {X 0,Y 376.572,Z 398.102,A -85,B 0,C 180,E1 -12883.01,E2 -12883.01} C_VEL
LIN {X 0,Y 374.518,Z 395.358,A -85,B 0,C 180,E1 -12883.833,E2 -12883.833} C_VEL
LIN {X 0,Y 373.643,Z 393.895,A -85,B 0,C 180,E1 -12884.153,E2 -12884.153} C_VEL
LIN {X 0,Y 370.851,Z 391.975,A -85,B 0,C 180,E1 -12885.068,E2 -12885.068} C_VEL
LIN {X 0,Y 369.451,Z 389.794,A -85,B 0,C 180,E1 -12885.569,E2 -12885.569} C_VEL
LIN {X 0,Y 369.036,Z 388.426,A -85,B 0,C 180,E1 -12885.888,E2 -12885.888} C_VEL
LIN {X 0,Y 368.971,Z 388.026,A -85,B 0,C 180,E1 -12886.601,E2 -12886.601} C_VEL
LIN {X 0,Y 368.932,Z 388.031,A -85,B 0,C 180,E1 -12890.053,E2 -12890.053} C_VEL
LIN {X 0,Y 368.94,Z 388.03,A -85,B 0,C 180,E1 -12893.887,E2 -12893.887} C_VEL
LIN {X 0,Y 368.966,Z 388.027,A -85,B 0,C 180,E1 -12897.203,E2 -12897.203} C_VEL
LIN {X 0,Y 368.917,Z 388.014,A -85,B 0,C 180,E1 -12899.689,E2 -12899.689} C_VEL
LIN {X 0,Y 368.89,Z 388.018,A -85,B 0,C 180,E1 -12903.538,E2 -12903.538} C_VEL
LIN {X 0,Y 368.901,Z 388.029,A -85,B 0,C 180,E1 -12906.857,E2 -12906.857} C_VEL
LIN {X 0,Y 368.946,Z 388.003,A -85,B 0,C 180,E1 -12910.364,E2 -12910.364} C_VEL
LIN {X 0,Y 368.876,Z 388.012,A -85,B 0,C 180,E1 -12913.616,E2 -12913.616} C_VEL
LIN {X 0,Y 368.896,Z 388.022,A -85,B 0,C 180,E1 -12914.772,E2 -12914.772} C_VEL
LIN {X 0,Y 368.284,Z 388.11,A -85,B 0,C 180,E1 -12915.683,E2 -12915.683} C_VEL
LIN {X 0,Y 365.436,Z 388.464,A -85,B 0,C 180,E1 -12917.164,E2 -12917.164} C_VEL
LIN {X 0,Y 362.99,Z 388.761,A -85,B 0,C 180,E1 -12918.362,E2 -12918.362} C_VEL
LIN {X 0,Y 361.941,Z 388.886,A -85,B 0,C 180,E1 -12919.289,E2 -12919.289} C_VEL
LIN {X 0,Y 361.858,Z 388.896,A -85,B 0,C 180,E1 -12919.603,E2 -12919.603} C_VEL
LIN {X 0,Y 361.866,Z 388.908,A -85,B 0,C 180,E1 -12922.983,E2 -12922.983} C_VEL
LIN {X 0,Y 361.852,Z 388.9,A -85,B 0,C 180,E1 -12926.631,E2 -12926.631} C_VEL
LIN {X 0,Y 361.871,Z 388.906,A -85,B 0,C 180,E1 -12929.673,E2 -12929.673} C_VEL
LIN {X 0,Y 361.948,Z 388.884,A -85,B 0,C 180,E1 -12933.475,E2 -12933.475} C_VEL
LIN {X 0,Y 361.883,Z 388.904,A -85,B 0,C 180,E1 -12937.145,E2 -12937.145} C_VEL
LIN {X 0,Y 361.9,Z 388.88,A -85,B 0,C 180,E1 -12940.724,E2 -12940.724} C_VEL
LIN {X 0,Y 361.926,Z 388.896,A -85,B 0,C 180,E1 -12943.066,E2 -12943.066} C_VEL
LIN {X 0,Y 361.993,Z 388.89,A -85,B 0,C 180,E1 -12946.528,E2 -12946.528} C_VEL
LIN {X 0,Y 362.027,Z 388.86,A -85,B 0,C 180,E1 -12949.939,E2 -12949.939} C_VEL
LIN {X 0,Y 362.145,Z 388.861,A -85,B 0,C 180,E1 -12952.193,E2 -12952.193} C_VEL
LIN {X 0,Y 362.113,Z 388.881,A -85,B 0,C 180,E1 -12954.432,E2 -12954.432} C_VEL
LIN {X 0,Y 362.277,Z 388.844,A -85,B 0,C 180,E1 -12957.777,E2 -12957.777} C_VEL
LIN {X 0,Y 362.422,Z 388.809,A -85,B 0,C 180,E1 -12960.001,E2 -12960.001} C_VEL
LIN {X 0,Y 362.278,Z 388.847,A -85,B 0,C 180,E1 -12962.224,E2 -12962.224} C_VEL
LIN {X 0,Y 362.167,Z 388.862,A -85,B 0,C 180,E1 -12966.687,E2 -12966.687} C_VEL
LIN {X 0,Y 362.069,Z 388.852,A -85,B 0,C 180,E1 -12968.934,E2 -12968.934} C_VEL
LIN {X 0,Y 361.955,Z 388.891,A -85,B 0,C 180,E1 -12972.333,E2 -12972.333} C_VEL
LIN {X 0,Y 361.959,Z 388.894,A -85,B 0,C 180,E1 -12974.621,E2 -12974.621} C_VEL
LIN {X 0,Y 361.952,Z 388.872,A -85,B 0,C 180,E1 -12978.1,E2 -12978.1} C_VEL
LIN {X 0,Y 361.888,Z 388.9,A -85,B 0,C 180,E1 -12981.654,E2 -12981.654} C_VEL
LIN {X 0,Y 361.925,Z 388.89,A -85,B 0,C 180,E1 -12985.291,E2 -12985.291} C_VEL
LIN {X 0,Y 361.919,Z 388.884,A -85,B 0,C 180,E1 -12987.779,E2 -12987.779} C_VEL
LIN {X 0,Y 361.857,Z 388.91,A -85,B 0,C 180,E1 -12991.628,E2 -12991.628} C_VEL
LIN {X 0,Y 361.872,Z 388.899,A -85,B 0,C 180,E1 -12995.346,E2 -12995.346} C_VEL
LIN {X 0,Y 361.873,Z 388.9,A -85,B 0,C 180,E1 -12999.029,E2 -12999.029} C_VEL
LIN {X 0,Y 361.888,Z 388.906,A -85,B 0,C 180,E1 -13002.442,E2 -13002.442} C_VEL
LIN {X 0,Y 361.846,Z 388.911,A -85,B 0,C 180,E1 -13005.637,E2 -13005.637} C_VEL
LIN {X 0,Y 361.834,Z 388.89,A -85,B 0,C 180,E1 -13009.246,E2 -13009.246} C_VEL
LIN {X 0,Y 361.865,Z 388.906,A -85,B 0,C 180,E1 -13012.778,E2 -13012.778} C_VEL
LIN {X 0,Y 361.856,Z 388.912,A -85,B 0,C 180,E1 -13015.721,E2 -13015.721} C_VEL
LIN {X 0,Y 361.945,Z 389.069,A -85,B 0,C 180,E1 -13018.382,E2 -13018.382} C_VEL
LIN {X 0,Y 363.483,Z 396.883,A -85,B 0,C 180,E1 -13021.094,E2 -13021.094} C_VEL
LIN {X 0,Y 364.986,Z 405.25,A -85,B 0,C 180,E1 -13023.713,E2 -13023.713} C_VEL
LIN {X 0,Y 364.548,Z 411.358,A -85,B 0,C 180,E1 -13025.513,E2 -13025.513} C_VEL
LIN {X 0,Y 363.737,Z 419.229,A -85,B 0,C 180,E1 -13027.841,E2 -13027.841} C_VEL
LIN {X 0,Y 364.736,Z 424.517,A -85,B 0,C 180,E1 -13028.068,E2 -13028.068} C_VEL
LIN {X 0,Y 369.524,Z 449.828,A -85,B 0,C 180,E1 -13028.881,E2 -13028.881} C_VEL
LIN {X 0,Y 370.15,Z 455.397,A -85,B 0,C 180,E1 -13029.031,E2 -13029.031} C_VEL
LIN {X 0,Y 368.997,Z 524.13,A -85,B 0,C 180,E1 -13030.386,E2 -13030.386} C_VEL
LIN {X 0,Y 368.614,Z 534.043,A -85,B 0,C 180,E1 -13030.691,E2 -13030.691} C_VEL
LIN {X 0,Y 367.976,Z 544.027,A -85,B 0,C 180,E1 -13031.126,E2 -13031.126} C_VEL
LIN {X 0,Y 367.212,Z 554.383,A -85,B 0,C 180,E1 -13031.736,E2 -13031.736} C_VEL
LIN {X 0,Y 366.435,Z 563.528,A -85,B 0,C 180,E1 -13032.418,E2 -13032.418} C_VEL
LIN {X 0,Y 365.521,Z 572.528,A -85,B 0,C 180,E1 -13033.238,E2 -13033.238} C_VEL
LIN {X 0,Y 364.664,Z 581.257,A -85,B 0,C 180,E1 -13034.204,E2 -13034.204} C_VEL
LIN {X 0,Y 363.846,Z 589.232,A -85,B 0,C 180,E1 -13035.257,E2 -13035.257} C_VEL
LIN {X 0,Y 362.977,Z 597.478,A -85,B 0,C 180,E1 -13036.565,E2 -13036.565} C_VEL
LIN {X 0,Y 362.276,Z 603.467,A -85,B 0,C 180,E1 -13037.679,E2 -13037.679} C_VEL
LIN {X 0,Y 361.586,Z 609.778,A -85,B 0,C 180,E1 -13039.076,E2 -13039.076} C_VEL
LIN {X 0,Y 361.084,Z 615.052,A -85,B 0,C 180,E1 -13040.478,E2 -13040.478} C_VEL
LIN {X 0,Y 360.673,Z 620.146,A -85,B 0,C 180,E1 -13042.161,E2 -13042.161} C_VEL
LIN {X 0,Y 360.5,Z 622.987,A -85,B 0,C 180,E1 -13043.283,E2 -13043.283} C_VEL
LIN {X 0,Y 360.35,Z 627.046,A -85,B 0,C 180,E1 -13045.526,E2 -13045.526} C_VEL
LIN {X 0,Y 360.298,Z 628.545,A -85,B 0,C 180,E1 -13046.646,E2 -13046.646} C_VEL
LIN {X 0,Y 360.303,Z 630.067,A -85,B 0,C 180,E1 -13048.883,E2 -13048.883} C_VEL
LIN {X 0,Y 360.343,Z 630.347,A -85,B 0,C 180,E1 -13050,E2 -13050} C_VEL
LIN {X 0,Y 360.265,Z 629.471,A -85,B 0,C 180,E1 -13052.236,E2 -13052.236} C_VEL
LIN {X 0,Y 360.298,Z 628.544,A -85,B 0,C 180,E1 -13053.355,E2 -13053.355} C_VEL
LIN {X 0,Y 360.365,Z 625.198,A -85,B 0,C 180,E1 -13055.596,E2 -13055.596} C_VEL
LIN {X 0,Y 360.594,Z 621.573,A -85,B 0,C 180,E1 -13057.278,E2 -13057.278} C_VEL
LIN {X 0,Y 360.932,Z 616.841,A -85,B 0,C 180,E1 -13058.962,E2 -13058.962} C_VEL
LIN {X 0,Y 361.507,Z 610.869,A -85,B 0,C 180,E1 -13060.643,E2 -13060.643} C_VEL
LIN {X 0,Y 361.939,Z 606.086,A -85,B 0,C 180,E1 -13061.764,E2 -13061.764} C_VEL
LIN {X 0,Y 362.605,Z 600.595,A -85,B 0,C 180,E1 -13062.879,E2 -13062.879} C_VEL
LIN {X 0,Y 363.497,Z 592.376,A -85,B 0,C 180,E1 -13064.271,E2 -13064.271} C_VEL
LIN {X 0,Y 364.226,Z 585.599,A -85,B 0,C 180,E1 -13065.249,E2 -13065.249} C_VEL
LIN {X 0,Y 365.166,Z 576.462,A -85,B 0,C 180,E1 -13066.348,E2 -13066.348} C_VEL
LIN {X 0,Y 366.14,Z 566.701,A -85,B 0,C 180,E1 -13067.309,E2 -13067.309} C_VEL
LIN {X 0,Y 366.937,Z 558.311,A -85,B 0,C 180,E1 -13067.99,E2 -13067.99} C_VEL
LIN {X 0,Y 367.697,Z 547.802,A -85,B 0,C 180,E1 -13068.672,E2 -13068.672} C_VEL
LIN {X 0,Y 368.415,Z 537.47,A -85,B 0,C 180,E1 -13069.176,E2 -13069.176} C_VEL
LIN {X 0,Y 368.93,Z 526.748,A -85,B 0,C 180,E1 -13069.546,E2 -13069.546} C_VEL
LIN {X 0,Y 369.386,Z 505.76,A -85,B 0,C 180,E1 -13069.991,E2 -13069.991} C_VEL
LIN {X 0,Y 370.094,Z 453,A -85,B 0,C 180,E1 -13071.021,E2 -13071.021} C_VEL
LIN {X 0,Y 365.018,Z 425.773,A -85,B 0,C 180,E1 -13071.888,E2 -13071.888} C_VEL
LIN {X 0,Y 363.701,Z 419.535,A -85,B 0,C 180,E1 -13072.127,E2 -13072.127} C_VEL
LIN {X 0,Y 363.689,Z 418.82,A -85,B 0,C 180,E1 -13072.24,E2 -13072.24} C_VEL
LIN {X 0,Y 365.005,Z 407.397,A -85,B 0,C 180,E1 -13075.672,E2 -13075.672} C_VEL
LIN {X 0,Y 364.751,Z 403.513,A -85,B 0,C 180,E1 -13076.879,E2 -13076.879} C_VEL
LIN {X 0,Y 363.059,Z 394.503,A -85,B 0,C 180,E1 -13079.767,E2 -13079.767} C_VEL
LIN {X 0,Y 361.919,Z 388.985,A -85,B 0,C 180,E1 -13081.703,E2 -13081.703} C_VEL
LIN {X 0,Y 361.871,Z 388.897,A -85,B 0,C 180,E1 -13085.636,E2 -13085.636} C_VEL
LIN {X 0,Y 361.873,Z 388.905,A -85,B 0,C 180,E1 -13089.026,E2 -13089.026} C_VEL
LIN {X 0,Y 361.84,Z 388.91,A -85,B 0,C 180,E1 -13092.828,E2 -13092.828} C_VEL
LIN {X 0,Y 361.914,Z 388.897,A -85,B 0,C 180,E1 -13095.931,E2 -13095.931} C_VEL
LIN {X 0,Y 361.908,Z 388.9,A -85,B 0,C 180,E1 -13099.231,E2 -13099.231} C_VEL
LIN {X 0,Y 361.874,Z 388.906,A -85,B 0,C 180,E1 -13102.982,E2 -13102.982} C_VEL
LIN {X 0,Y 361.863,Z 388.896,A -85,B 0,C 180,E1 -13106.629,E2 -13106.629} C_VEL
LIN {X 0,Y 361.877,Z 388.91,A -85,B 0,C 180,E1 -13109.672,E2 -13109.672} C_VEL
LIN {X 0,Y 361.955,Z 388.876,A -85,B 0,C 180,E1 -13113.475,E2 -13113.475} C_VEL
LIN {X 0,Y 361.89,Z 388.903,A -85,B 0,C 180,E1 -13117.144,E2 -13117.144} C_VEL
LIN {X 0,Y 361.906,Z 388.881,A -85,B 0,C 180,E1 -13120.723,E2 -13120.723} C_VEL
LIN {X 0,Y 361.934,Z 388.883,A -85,B 0,C 180,E1 -13123.065,E2 -13123.065} C_VEL
LIN {X 0,Y 361.998,Z 388.888,A -85,B 0,C 180,E1 -13126.527,E2 -13126.527} C_VEL
LIN {X 0,Y 362.03,Z 388.857,A -85,B 0,C 180,E1 -13129.937,E2 -13129.937} C_VEL
LIN {X 0,Y 362.145,Z 388.856,A -85,B 0,C 180,E1 -13132.192,E2 -13132.192} C_VEL
LIN {X 0,Y 362.117,Z 388.875,A -85,B 0,C 180,E1 -13134.431,E2 -13134.431} C_VEL
LIN {X 0,Y 362.281,Z 388.847,A -85,B 0,C 180,E1 -13137.776,E2 -13137.776} C_VEL
LIN {X 0,Y 362.424,Z 388.808,A -85,B 0,C 180,E1 -13139.999,E2 -13139.999} C_VEL
LIN {X 0,Y 362.281,Z 388.843,A -85,B 0,C 180,E1 -13142.223,E2 -13142.223} C_VEL
LIN {X 0,Y 362.17,Z 388.867,A -85,B 0,C 180,E1 -13146.686,E2 -13146.686} C_VEL
LIN {X 0,Y 362.073,Z 388.863,A -85,B 0,C 180,E1 -13148.933,E2 -13148.933} C_VEL
LIN {X 0,Y 361.964,Z 388.888,A -85,B 0,C 180,E1 -13152.332,E2 -13152.332} C_VEL
LIN {X 0,Y 361.96,Z 388.895,A -85,B 0,C 180,E1 -13154.62,E2 -13154.62} C_VEL
LIN {X 0,Y 361.953,Z 388.878,A -85,B 0,C 180,E1 -13158.099,E2 -13158.099} C_VEL
LIN {X 0,Y 361.889,Z 388.9,A -85,B 0,C 180,E1 -13161.652,E2 -13161.652} C_VEL
LIN {X 0,Y 361.925,Z 388.896,A -85,B 0,C 180,E1 -13165.29,E2 -13165.29} C_VEL
LIN {X 0,Y 361.905,Z 388.885,A -85,B 0,C 180,E1 -13167.779,E2 -13167.779} C_VEL
LIN {X 0,Y 361.834,Z 388.914,A -85,B 0,C 180,E1 -13171.629,E2 -13171.629} C_VEL
LIN {X 0,Y 361.871,Z 388.894,A -85,B 0,C 180,E1 -13175.344,E2 -13175.344} C_VEL
LIN {X 0,Y 361.868,Z 388.908,A -85,B 0,C 180,E1 -13179.027,E2 -13179.027} C_VEL
LIN {X 0,Y 361.833,Z 388.911,A -85,B 0,C 180,E1 -13182.828,E2 -13182.828} C_VEL
LIN {X 0,Y 361.817,Z 388.897,A -85,B 0,C 180,E1 -13185.946,E2 -13185.946} C_VEL
LIN {X 0,Y 361.864,Z 388.877,A -85,B 0,C 180,E1 -13189.238,E2 -13189.238} C_VEL
LIN {X 0,Y 361.874,Z 388.906,A -85,B 0,C 180,E1 -13192.983,E2 -13192.983} C_VEL
LIN {X 0,Y 361.855,Z 388.896,A -85,B 0,C 180,E1 -13196.63,E2 -13196.63} C_VEL
LIN {X 0,Y 361.873,Z 388.897,A -85,B 0,C 180,E1 -13199.672,E2 -13199.672} C_VEL
LIN {X 0,Y 361.951,Z 388.901,A -85,B 0,C 180,E1 -13203.475,E2 -13203.475} C_VEL
LIN {X 0,Y 361.887,Z 388.909,A -85,B 0,C 180,E1 -13207.144,E2 -13207.144} C_VEL
LIN {X 0,Y 361.917,Z 388.905,A -85,B 0,C 180,E1 -13210.724,E2 -13210.724} C_VEL
LIN {X 0,Y 361.991,Z 389.166,A -85,B 0,C 180,E1 -13212.265,E2 -13212.265} C_VEL
LIN {X 0,Y 362.282,Z 390.407,A -85,B 0,C 180,E1 -13212.581,E2 -13212.581} C_VEL
LIN {X 0,Y 363.83,Z 392.9,A -85,B 0,C 180,E1 -13213.063,E2 -13213.063} C_VEL
LIN {X 0,Y 366.435,Z 394.936,A -85,B 0,C 180,E1 -13213.835,E2 -13213.835} C_VEL
LIN {X 0,Y 368.239,Z 397.826,A -85,B 0,C 180,E1 -13214.424,E2 -13214.424} C_VEL
LIN {X 0,Y 371.016,Z 400.143,A -85,B 0,C 180,E1 -13215.323,E2 -13215.323} C_VEL
LIN {X 0,Y 371.854,Z 400.825,A -85,B 0,C 180,E1 -13215.602,E2 -13215.602} C_VEL
LIN {X 0,Y 374.175,Z 404.028,A -85,B 0,C 180,E1 -13216.444,E2 -13216.444} C_VEL
LIN {X 0,Y 376.963,Z 406.259,A -85,B 0,C 180,E1 -13217.483,E2 -13217.483} C_VEL
LIN {X 0,Y 377.928,Z 407.045,A -85,B 0,C 180,E1 -13217.856,E2 -13217.856} C_VEL
LIN {X 0,Y 380.531,Z 410.379,A -85,B 0,C 180,E1 -13219.02,E2 -13219.02} C_VEL
LIN {X 0,Y 383.373,Z 412.5,A -85,B 0,C 180,E1 -13220.37,E2 -13220.37} C_VEL
LIN {X 0,Y 384.988,Z 413.442,A -85,B 0,C 180,E1 -13221.206,E2 -13221.206} C_VEL
LIN {X 0,Y 387.165,Z 416.425,A -85,B 0,C 180,E1 -13222.596,E2 -13222.596} C_VEL
LIN {X 0,Y 389.393,Z 418.395,A -85,B 0,C 180,E1 -13224.303,E2 -13224.303} C_VEL
LIN {X 0,Y 391.009,Z 419.284,A -85,B 0,C 180,E1 -13225.877,E2 -13225.877} C_VEL
LIN {X 0,Y 392.127,Z 419.662,A -85,B 0,C 180,E1 -13227.45,E2 -13227.45} C_VEL
LIN {X 0,Y 392.684,Z 420.085,A -85,B 0,C 180,E1 -13228.974,E2 -13228.974} C_VEL
LIN {X 0,Y 392.864,Z 420.023,A -85,B 0,C 180,E1 -13230,E2 -13230} C_VEL
LIN {X 0,Y 392.598,Z 419.972,A -85,B 0,C 180,E1 -13231.538,E2 -13231.538} C_VEL
LIN {X 0,Y 391.863,Z 419.545,A -85,B 0,C 180,E1 -13233.084,E2 -13233.084} C_VEL
LIN {X 0,Y 390.284,Z 418.938,A -85,B 0,C 180,E1 -13234.906,E2 -13234.906} C_VEL
LIN {X 0,Y 388.217,Z 417.454,A -85,B 0,C 180,E1 -13236.635,E2 -13236.635} C_VEL
LIN {X 0,Y 386.33,Z 415.399,A -85,B 0,C 180,E1 -13237.961,E2 -13237.961} C_VEL
LIN {X 0,Y 384.776,Z 413.129,A -85,B 0,C 180,E1 -13238.931,E2 -13238.931} C_VEL
LIN {X 0,Y 381.794,Z 411.494,A -85,B 0,C 180,E1 -13240.39,E2 -13240.39} C_VEL
LIN {X 0,Y 379.123,Z 408.829,A -85,B 0,C 180,E1 -13241.589,E2 -13241.589} C_VEL
LIN {X 0,Y 377.389,Z 406.466,A -85,B 0,C 180,E1 -13242.366,E2 -13242.366} C_VEL
LIN {X 0,Y 374.536,Z 404.423,A -85,B 0,C 180,E1 -13243.414,E2 -13243.414} C_VEL
LIN {X 0,Y 372.156,Z 401.361,A -85,B 0,C 180,E1 -13244.288,E2 -13244.288} C_VEL
LIN {X 0,Y 371.417,Z 400.381,A -85,B 0,C 180,E1 -13244.548,E2 -13244.548} C_VEL
LIN {X 0,Y 368.757,Z 398.335,A -85,B 0,C 180,E1 -13245.421,E2 -13245.421} C_VEL
LIN {X 0,Y 366.786,Z 395.692,A -85,B 0,C 180,E1 -13246.042,E2 -13246.042} C_VEL
LIN {X 0,Y 366.071,Z 394.535,A -85,B 0,C 180,E1 -13246.279,E2 -13246.279} C_VEL
LIN {X 0,Y 363.706,Z 392.787,A -85,B 0,C 180,E1 -13246.969,E2 -13246.969} C_VEL
LIN {X 0,Y 362.154,Z 389.988,A -85,B 0,C 180,E1 -13247.489,E2 -13247.489} C_VEL
LIN {X 0,Y 361.958,Z 389.007,A -85,B 0,C 180,E1 -13247.859,E2 -13247.859} C_VEL
LIN {X 0,Y 361.887,Z 388.909,A -85,B 0,C 180,E1 -13251.653,E2 -13251.653} C_VEL
LIN {X 0,Y 361.923,Z 388.904,A -85,B 0,C 180,E1 -13255.29,E2 -13255.29} C_VEL
LIN {X 0,Y 361.917,Z 388.901,A -85,B 0,C 180,E1 -13257.778,E2 -13257.778} C_VEL
LIN {X 0,Y 361.841,Z 388.914,A -85,B 0,C 180,E1 -13261.285,E2 -13261.285} C_VEL
LIN {X 0,Y 361.848,Z 388.886,A -85,B 0,C 180,E1 -13264.28,E2 -13264.28} C_VEL
LIN {X 0,Y 361.87,Z 388.91,A -85,B 0,C 180,E1 -13267.225,E2 -13267.225} C_VEL
LIN {X 0,Y 361.861,Z 388.878,A -85,B 0,C 180,E1 -13270.761,E2 -13270.761} C_VEL
LIN {X 0,Y 361.828,Z 388.898,A -85,B 0,C 180,E1 -13274.366,E2 -13274.366} C_VEL
LIN {X 0,Y 361.85,Z 388.908,A -85,B 0,C 180,E1 -13277.564,E2 -13277.564} C_VEL
LIN {X 0,Y 361.858,Z 388.896,A -85,B 0,C 180,E1 -13279.603,E2 -13279.603} C_VEL
LIN {X 0,Y 361.2,Z 388.986,A -85,B 0,C 180,E1 -13280.532,E2 -13280.532} C_VEL
LIN {X 0,Y 358.357,Z 389.346,A -85,B 0,C 180,E1 -13282.042,E2 -13282.042} C_VEL
LIN {X 0,Y 355.94,Z 389.645,A -85,B 0,C 180,E1 -13283.264,E2 -13283.264} C_VEL
LIN {X 0,Y 354.895,Z 389.769,A -85,B 0,C 180,E1 -13284.209,E2 -13284.209} C_VEL
LIN {X 0,Y 354.807,Z 389.775,A -85,B 0,C 180,E1 -13284.529,E2 -13284.529} C_VEL
LIN {X 0,Y 354.78,Z 389.788,A -85,B 0,C 180,E1 -13287.667,E2 -13287.667} C_VEL
LIN {X 0,Y 354.862,Z 389.774,A -85,B 0,C 180,E1 -13290.621,E2 -13290.621} C_VEL
LIN {X 0,Y 354.892,Z 389.765,A -85,B 0,C 180,E1 -13294.173,E2 -13294.173} C_VEL
LIN {X 0,Y 354.828,Z 389.783,A -85,B 0,C 180,E1 -13297.894,E2 -13297.894} C_VEL
LIN {X 0,Y 354.916,Z 389.754,A -85,B 0,C 180,E1 -13301.892,E2 -13301.892} C_VEL
LIN {X 0,Y 354.937,Z 389.772,A -85,B 0,C 180,E1 -13305.981,E2 -13305.981} C_VEL
LIN {X 0,Y 354.974,Z 389.738,A -85,B 0,C 180,E1 -13309.736,E2 -13309.736} C_VEL
LIN {X 0,Y 355.108,Z 389.736,A -85,B 0,C 180,E1 -13312.037,E2 -13312.037} C_VEL
LIN {X 0,Y 355.087,Z 389.755,A -85,B 0,C 180,E1 -13314.321,E2 -13314.321} C_VEL
LIN {X 0,Y 355.241,Z 389.72,A -85,B 0,C 180,E1 -13317.733,E2 -13317.733} C_VEL
LIN {X 0,Y 355.371,Z 389.686,A -85,B 0,C 180,E1 -13320.001,E2 -13320.001} C_VEL
LIN {X 0,Y 355.241,Z 389.724,A -85,B 0,C 180,E1 -13322.268,E2 -13322.268} C_VEL
LIN {X 0,Y 355.132,Z 389.737,A -85,B 0,C 180,E1 -13326.82,E2 -13326.82} C_VEL
LIN {X 0,Y 355.01,Z 389.73,A -85,B 0,C 180,E1 -13329.113,E2 -13329.113} C_VEL
LIN {X 0,Y 354.916,Z 389.771,A -85,B 0,C 180,E1 -13332.582,E2 -13332.582} C_VEL
LIN {X 0,Y 354.887,Z 389.768,A -85,B 0,C 180,E1 -13336.097,E2 -13336.097} C_VEL
LIN {X 0,Y 354.897,Z 389.749,A -85,B 0,C 180,E1 -13338.473,E2 -13338.473} C_VEL
LIN {X 0,Y 354.831,Z 389.783,A -85,B 0,C 180,E1 -13342.107,E2 -13342.107} C_VEL
LIN {X 0,Y 354.896,Z 389.759,A -85,B 0,C 180,E1 -13345.828,E2 -13345.828} C_VEL
LIN {X 0,Y 354.852,Z 389.78,A -85,B 0,C 180,E1 -13349.679,E2 -13349.679} C_VEL
LIN {X 0,Y 354.828,Z 389.77,A -85,B 0,C 180,E1 -13353.683,E2 -13353.683} C_VEL
LIN {X 0,Y 354.8,Z 389.79,A -85,B 0,C 180,E1 -13356.46,E2 -13356.46} C_VEL
LIN {X 0,Y 354.822,Z 389.777,A -85,B 0,C 180,E1 -13359.425,E2 -13359.425} C_VEL
LIN {X 0,Y 354.837,Z 389.782,A -85,B 0,C 180,E1 -13362.877,E2 -13362.877} C_VEL
LIN {X 0,Y 354.783,Z 389.795,A -85,B 0,C 180,E1 -13366.107,E2 -13366.107} C_VEL
LIN {X 0,Y 354.787,Z 389.767,A -85,B 0,C 180,E1 -13369.18,E2 -13369.18} C_VEL
LIN {X 0,Y 354.808,Z 389.787,A -85,B 0,C 180,E1 -13372.403,E2 -13372.403} C_VEL
LIN {X 0,Y 354.813,Z 389.779,A -85,B 0,C 180,E1 -13374.942,E2 -13374.942} C_VEL
LIN {X 0,Y 354.883,Z 389.962,A -85,B 0,C 180,E1 -13378.028,E2 -13378.028} C_VEL
LIN {X 0,Y 356.443,Z 397.739,A -85,B 0,C 180,E1 -13380.792,E2 -13380.792} C_VEL
LIN {X 0,Y 357.978,Z 406.11,A -85,B 0,C 180,E1 -13383.473,E2 -13383.473} C_VEL
LIN {X 0,Y 357.899,Z 409.802,A -85,B 0,C 180,E1 -13384.596,E2 -13384.596} C_VEL
LIN {X 0,Y 356.834,Z 418.995,A -85,B 0,C 180,E1 -13387.381,E2 -13387.381} C_VEL
LIN {X 0,Y 357.669,Z 423.302,A -85,B 0,C 180,E1 -13387.59,E2 -13387.59} C_VEL
LIN {X 0,Y 362.767,Z 449.764,A -85,B 0,C 180,E1 -13388.471,E2 -13388.471} C_VEL
LIN {X 0,Y 363.542,Z 454.997,A -85,B 0,C 180,E1 -13388.627,E2 -13388.627} C_VEL
LIN {X 0,Y 362.324,Z 523.94,A -85,B 0,C 180,E1 -13390.01,E2 -13390.01} C_VEL
LIN {X 0,Y 361.907,Z 533.848,A -85,B 0,C 180,E1 -13390.318,E2 -13390.318} C_VEL
LIN {X 0,Y 361.272,Z 543.832,A -85,B 0,C 180,E1 -13390.763,E2 -13390.763} C_VEL
LIN {X 0,Y 360.454,Z 554.187,A -85,B 0,C 180,E1 -13391.382,E2 -13391.382} C_VEL
LIN {X 0,Y 359.65,Z 563.332,A -85,B 0,C 180,E1 -13392.075,E2 -13392.075} C_VEL
LIN {X 0,Y 358.723,Z 572.333,A -85,B 0,C 180,E1 -13392.91,E2 -13392.91} C_VEL
LIN {X 0,Y 357.824,Z 581.061,A -85,B 0,C 180,E1 -13393.894,E2 -13393.894} C_VEL
LIN {X 0,Y 357.013,Z 588.499,A -85,B 0,C 180,E1 -13394.883,E2 -13394.883} C_VEL
LIN {X 0,Y 356.034,Z 597.281,A -85,B 0,C 180,E1 -13396.298,E2 -13396.298} C_VEL
LIN {X 0,Y 355.319,Z 603.271,A -85,B 0,C 180,E1 -13397.434,E2 -13397.434} C_VEL
LIN {X 0,Y 354.579,Z 609.582,A -85,B 0,C 180,E1 -13398.858,E2 -13398.858} C_VEL
LIN {X 0,Y 354.049,Z 614.856,A -85,B 0,C 180,E1 -13400.287,E2 -13400.287} C_VEL
LIN {X 0,Y 353.617,Z 619.951,A -85,B 0,C 180,E1 -13402.003,E2 -13402.003} C_VEL
LIN {X 0,Y 353.419,Z 622.791,A -85,B 0,C 180,E1 -13403.148,E2 -13403.148} C_VEL
LIN {X 0,Y 353.265,Z 626.85,A -85,B 0,C 180,E1 -13405.436,E2 -13405.436} C_VEL
LIN {X 0,Y 353.219,Z 628.35,A -85,B 0,C 180,E1 -13406.578,E2 -13406.578} C_VEL
LIN {X 0,Y 353.203,Z 629.872,A -85,B 0,C 180,E1 -13408.86,E2 -13408.86} C_VEL
LIN {X 0,Y 353.246,Z 630.152,A -85,B 0,C 180,E1 -13410,E2 -13410} C_VEL
LIN {X 0,Y 353.173,Z 629.276,A -85,B 0,C 180,E1 -13412.281,E2 -13412.281} C_VEL
LIN {X 0,Y 353.219,Z 628.349,A -85,B 0,C 180,E1 -13413.422,E2 -13413.422} C_VEL
LIN {X 0,Y 353.284,Z 625.002,A -85,B 0,C 180,E1 -13415.709,E2 -13415.709} C_VEL
LIN {X 0,Y 353.517,Z 621.377,A -85,B 0,C 180,E1 -13417.425,E2 -13417.425} C_VEL
LIN {X 0,Y 353.89,Z 616.645,A -85,B 0,C 180,E1 -13419.142,E2 -13419.142} C_VEL
LIN {X 0,Y 354.472,Z 610.672,A -85,B 0,C 180,E1 -13420.857,E2 -13420.857} C_VEL
LIN {X 0,Y 355.141,Z 604.579,A -85,B 0,C 180,E1 -13422.283,E2 -13422.283} C_VEL
LIN {X 0,Y 355.859,Z 598.839,A -85,B 0,C 180,E1 -13423.418,E2 -13423.418} C_VEL
LIN {X 0,Y 356.606,Z 592.181,A -85,B 0,C 180,E1 -13424.553,E2 -13424.553} C_VEL
LIN {X 0,Y 357.546,Z 583.701,A -85,B 0,C 180,E1 -13425.767,E2 -13425.767} C_VEL
LIN {X 0,Y 358.338,Z 576.267,A -85,B 0,C 180,E1 -13426.669,E2 -13426.669} C_VEL
LIN {X 0,Y 359.36,Z 566.505,A -85,B 0,C 180,E1 -13427.646,E2 -13427.646} C_VEL
LIN {X 0,Y 360.175,Z 558.115,A -85,B 0,C 180,E1 -13428.339,E2 -13428.339} C_VEL
LIN {X 0,Y 360.98,Z 547.607,A -85,B 0,C 180,E1 -13429.033,E2 -13429.033} C_VEL
LIN {X 0,Y 361.729,Z 537.276,A -85,B 0,C 180,E1 -13429.545,E2 -13429.545} C_VEL
LIN {X 0,Y 362.264,Z 526.554,A -85,B 0,C 180,E1 -13429.921,E2 -13429.921} C_VEL
LIN {X 0,Y 362.702,Z 503.773,A -85,B 0,C 180,E1 -13430.413,E2 -13430.413} C_VEL
LIN {X 0,Y 363.413,Z 453.8,A -85,B 0,C 180,E1 -13431.406,E2 -13431.406} C_VEL
LIN {X 0,Y 358.383,Z 426.7,A -85,B 0,C 180,E1 -13432.291,E2 -13432.291} C_VEL
LIN {X 0,Y 356.828,Z 419.195,A -85,B 0,C 180,E1 -13432.59,E2 -13432.59} C_VEL
LIN {X 0,Y 356.988,Z 416.985,A -85,B 0,C 180,E1 -13433.187,E2 -13433.187} C_VEL
LIN {X 0,Y 358.115,Z 407.204,A -85,B 0,C 180,E1 -13436.204,E2 -13436.204} C_VEL
LIN {X 0,Y 356.746,Z 399.102,A -85,B 0,C 180,E1 -13438.859,E2 -13438.859} C_VEL
LIN {X 0,Y 354.866,Z 389.876,A -85,B 0,C 180,E1 -13442.024,E2 -13442.024} C_VEL
LIN {X 0,Y 354.825,Z 389.773,A -85,B 0,C 180,E1 -13445.699,E2 -13445.699} C_VEL
LIN {X 0,Y 354.826,Z 389.773,A -85,B 0,C 180,E1 -13449.423,E2 -13449.423} C_VEL
LIN {X 0,Y 354.792,Z 389.788,A -85,B 0,C 180,E1 -13452.867,E2 -13452.867} C_VEL
LIN {X 0,Y 354.854,Z 389.777,A -85,B 0,C 180,E1 -13456.116,E2 -13456.116} C_VEL
LIN {X 0,Y 354.859,Z 389.778,A -85,B 0,C 180,E1 -13459.188,E2 -13459.188} C_VEL
LIN {X 0,Y 354.814,Z 389.788,A -85,B 0,C 180,E1 -13462.401,E2 -13462.401} C_VEL
LIN {X 0,Y 354.814,Z 389.778,A -85,B 0,C 180,E1 -13464.94,E2 -13464.94} C_VEL
LIN {X 0,Y 354.815,Z 389.787,A -85,B 0,C 180,E1 -13468.399,E2 -13468.399} C_VEL
LIN {X 0,Y 354.854,Z 389.771,A -85,B 0,C 180,E1 -13471.619,E2 -13471.619} C_VEL
LIN {X 0,Y 354.9,Z 389.759,A -85,B 0,C 180,E1 -13474.172,E2 -13474.172} C_VEL
LIN {X 0,Y 354.835,Z 389.783,A -85,B 0,C 180,E1 -13477.893,E2 -13477.893} C_VEL
LIN {X 0,Y 354.922,Z 389.747,A -85,B 0,C 180,E1 -13481.891,E2 -13481.891} C_VEL
LIN {X 0,Y 354.942,Z 389.77,A -85,B 0,C 180,E1 -13485.98,E2 -13485.98} C_VEL
LIN {X 0,Y 354.977,Z 389.737,A -85,B 0,C 180,E1 -13489.735,E2 -13489.735} C_VEL
LIN {X 0,Y 355.127,Z 389.726,A -85,B 0,C 180,E1 -13492.037,E2 -13492.037} C_VEL
LIN {X 0,Y 355.091,Z 389.751,A -85,B 0,C 180,E1 -13494.32,E2 -13494.32} C_VEL
LIN {X 0,Y 355.244,Z 389.724,A -85,B 0,C 180,E1 -13497.732,E2 -13497.732} C_VEL
LIN {X 0,Y 355.373,Z 389.686,A -85,B 0,C 180,E1 -13499.999,E2 -13499.999} C_VEL
LIN {X 0,Y 355.244,Z 389.72,A -85,B 0,C 180,E1 -13502.267,E2 -13502.267} C_VEL
LIN {X 0,Y 355.136,Z 389.743,A -85,B 0,C 180,E1 -13506.819,E2 -13506.819} C_VEL
LIN {X 0,Y 355.014,Z 389.739,A -85,B 0,C 180,E1 -13509.112,E2 -13509.112} C_VEL
LIN {X 0,Y 354.923,Z 389.765,A -85,B 0,C 180,E1 -13512.58,E2 -13512.58} C_VEL
LIN {X 0,Y 354.887,Z 389.773,A -85,B 0,C 180,E1 -13516.095,E2 -13516.095} C_VEL
LIN {X 0,Y 354.898,Z 389.755,A -85,B 0,C 180,E1 -13518.472,E2 -13518.472} C_VEL
LIN {X 0,Y 354.832,Z 389.783,A -85,B 0,C 180,E1 -13522.105,E2 -13522.105} C_VEL
LIN {X 0,Y 354.896,Z 389.765,A -85,B 0,C 180,E1 -13525.827,E2 -13525.827} C_VEL
LIN {X 0,Y 354.814,Z 389.784,A -85,B 0,C 180,E1 -13529.681,E2 -13529.681} C_VEL
LIN {X 0,Y 354.803,Z 389.774,A -85,B 0,C 180,E1 -13533.702,E2 -13533.702} C_VEL
LIN {X 0,Y 354.798,Z 389.785,A -85,B 0,C 180,E1 -13536.459,E2 -13536.459} C_VEL
LIN {X 0,Y 354.82,Z 389.78,A -85,B 0,C 180,E1 -13539.423,E2 -13539.423} C_VEL
LIN {X 0,Y 354.786,Z 389.789,A -85,B 0,C 180,E1 -13542.867,E2 -13542.867} C_VEL
LIN {X 0,Y 354.765,Z 389.773,A -85,B 0,C 180,E1 -13546.104,E2 -13546.104} C_VEL
LIN {X 0,Y 354.815,Z 389.753,A -85,B 0,C 180,E1 -13549.183,E2 -13549.183} C_VEL
LIN {X 0,Y 354.812,Z 389.788,A -85,B 0,C 180,E1 -13552.4,E2 -13552.4} C_VEL
LIN {X 0,Y 354.808,Z 389.763,A -85,B 0,C 180,E1 -13554.94,E2 -13554.94} C_VEL
LIN {X 0,Y 354.79,Z 389.791,A -85,B 0,C 180,E1 -13558.405,E2 -13558.405} C_VEL
LIN {X 0,Y 354.85,Z 389.77,A -85,B 0,C 180,E1 -13561.619,E2 -13561.619} C_VEL
LIN {X 0,Y 354.896,Z 389.779,A -85,B 0,C 180,E1 -13564.172,E2 -13564.172} C_VEL
LIN {X 0,Y 354.831,Z 389.788,A -85,B 0,C 180,E1 -13567.894,E2 -13567.894} C_VEL
LIN {X 0,Y 354.913,Z 390.03,A -85,B 0,C 180,E1 -13570.666,E2 -13570.666} C_VEL
LIN {X 0,Y 355.228,Z 391.267,A -85,B 0,C 180,E1 -13570.969,E2 -13570.969} C_VEL
LIN {X 0,Y 356.952,Z 393.981,A -85,B 0,C 180,E1 -13571.466,E2 -13571.466} C_VEL
LIN {X 0,Y 359.108,Z 395.666,A -85,B 0,C 180,E1 -13572.017,E2 -13572.017} C_VEL
LIN {X 0,Y 361.066,Z 398.812,A -85,B 0,C 180,E1 -13572.61,E2 -13572.61} C_VEL
LIN {X 0,Y 364.12,Z 401.418,A -85,B 0,C 180,E1 -13573.452,E2 -13573.452} C_VEL
LIN {X 0,Y 366.387,Z 404.546,A -85,B 0,C 180,E1 -13574.187,E2 -13574.187} C_VEL
LIN {X 0,Y 369.303,Z 406.873,A -85,B 0,C 180,E1 -13575.083,E2 -13575.083} C_VEL
LIN {X 0,Y 370.76,Z 408.79,A -85,B 0,C 180,E1 -13575.602,E2 -13575.602} C_VEL
LIN {X 0,Y 373.643,Z 411.809,A -85,B 0,C 180,E1 -13576.619,E2 -13576.619} C_VEL
LIN {X 0,Y 376.096,Z 413.585,A -85,B 0,C 180,E1 -13577.522,E2 -13577.522} C_VEL
LIN {X 0,Y 378.785,Z 416.887,A -85,B 0,C 180,E1 -13578.686,E2 -13578.686} C_VEL
LIN {X 0,Y 381.522,Z 419.084,A -85,B 0,C 180,E1 -13579.929,E2 -13579.929} C_VEL
LIN {X 0,Y 383.693,Z 420.292,A -85,B 0,C 180,E1 -13580.976,E2 -13580.976} C_VEL
LIN {X 0,Y 386.24,Z 423.58,A -85,B 0,C 180,E1 -13582.578,E2 -13582.578} C_VEL
LIN {X 0,Y 388.479,Z 425.42,A -85,B 0,C 180,E1 -13584.266,E2 -13584.266} C_VEL
LIN {X 0,Y 390.135,Z 426.322,A -85,B 0,C 180,E1 -13585.868,E2 -13585.868} C_VEL
LIN {X 0,Y 391.261,Z 426.709,A -85,B 0,C 180,E1 -13587.445,E2 -13587.445} C_VEL
LIN {X 0,Y 391.823,Z 427.132,A -85,B 0,C 180,E1 -13588.972,E2 -13588.972} C_VEL
LIN {X 0,Y 391.999,Z 427.07,A -85,B 0,C 180,E1 -13590,E2 -13590} C_VEL
LIN {X 0,Y 391.73,Z 427.019,A -85,B 0,C 180,E1 -13591.542,E2 -13591.542} C_VEL
LIN {X 0,Y 390.988,Z 426.591,A -85,B 0,C 180,E1 -13593.091,E2 -13593.091} C_VEL
LIN {X 0,Y 389.394,Z 425.983,A -85,B 0,C 180,E1 -13594.918,E2 -13594.918} C_VEL
LIN {X 0,Y 387.299,Z 424.538,A -85,B 0,C 180,E1 -13596.653,E2 -13596.653} C_VEL
LIN {X 0,Y 385.253,Z 422.477,A -85,B 0,C 180,E1 -13598.051,E2 -13598.051} C_VEL
LIN {X 0,Y 383.437,Z 420.01,A -85,B 0,C 180,E1 -13599.167,E2 -13599.167} C_VEL
LIN {X 0,Y 380.179,Z 418.119,A -85,B 0,C 180,E1 -13600.72,E2 -13600.72} C_VEL
LIN {X 0,Y 376.999,Z 414.845,A -85,B 0,C 180,E1 -13602.106,E2 -13602.106} C_VEL
LIN {X 0,Y 375.689,Z 413.212,A -85,B 0,C 180,E1 -13602.629,E2 -13602.629} C_VEL
LIN {X 0,Y 372.562,Z 410.813,A -85,B 0,C 180,E1 -13603.783,E2 -13603.783} C_VEL
LIN {X 0,Y 369.83,Z 407.411,A -85,B 0,C 180,E1 -13604.735,E2 -13604.735} C_VEL
LIN {X 0,Y 366.128,Z 404.291,A -85,B 0,C 180,E1 -13605.892,E2 -13605.892} C_VEL
LIN {X 0,Y 363.96,Z 401.139,A -85,B 0,C 180,E1 -13606.602,E2 -13606.602} C_VEL
LIN {X 0,Y 361.065,Z 398.833,A -85,B 0,C 180,E1 -13607.39,E2 -13607.39} C_VEL
LIN {X 0,Y 358.715,Z 395.224,A -85,B 0,C 180,E1 -13608.097,E2 -13608.097} C_VEL
LIN {X 0,Y 356.346,Z 393.314,A -85,B 0,C 180,E1 -13608.688,E2 -13608.688} C_VEL
LIN {X 0,Y 355.026,Z 390.608,A -85,B 0,C 180,E1 -13609.139,E2 -13609.139} C_VEL
LIN {X 0,Y 354.859,Z 389.836,A -85,B 0,C 180,E1 -13609.524,E2 -13609.524} C_VEL
LIN {X 0,Y 354.827,Z 389.788,A -85,B 0,C 180,E1 -13613.336,E2 -13613.336} C_VEL
LIN {X 0,Y 354.884,Z 389.782,A -85,B 0,C 180,E1 -13616.982,E2 -13616.982} C_VEL
LIN {X 0,Y 354.849,Z 389.765,A -85,B 0,C 180,E1 -13619.678,E2 -13619.678} C_VEL
LIN {X 0,Y 354.8,Z 389.768,A -85,B 0,C 180,E1 -13623.702,E2 -13623.702} C_VEL
LIN {X 0,Y 354.798,Z 389.78,A -85,B 0,C 180,E1 -13626.458,E2 -13626.458} C_VEL
LIN {X 0,Y 354.819,Z 389.779,A -85,B 0,C 180,E1 -13629.424,E2 -13629.424} C_VEL
LIN {X 0,Y 354.784,Z 389.752,A -85,B 0,C 180,E1 -13632.868,E2 -13632.868} C_VEL
LIN {X 0,Y 354.778,Z 389.79,A -85,B 0,C 180,E1 -13636.106,E2 -13636.106} C_VEL
LIN {X 0,Y 354.795,Z 389.775,A -85,B 0,C 180,E1 -13639.598,E2 -13639.598} C_VEL
LIN {X 0,Y 354.806,Z 389.792,A -85,B 0,C 180,E1 -13642.401,E2 -13642.401} C_VEL
LIN {X 0,Y 354.807,Z 389.775,A -85,B 0,C 180,E1 -13644.529,E2 -13644.529} C_VEL
LIN {X 0,Y 354.117,Z 389.858,A -85,B 0,C 180,E1 -13645.476,E2 -13645.476} C_VEL
LIN {X 0,Y 351.221,Z 390.23,A -85,B 0,C 180,E1 -13647.016,E2 -13647.016} C_VEL
LIN {X 0,Y 348.805,Z 390.536,A -85,B 0,C 180,E1 -13648.262,E2 -13648.262} C_VEL
LIN {X 0,Y 347.809,Z 390.659,A -85,B 0,C 180,E1 -13649.227,E2 -13649.227} C_VEL
LIN {X 0,Y 347.75,Z 390.665,A -85,B 0,C 180,E1 -13649.553,E2 -13649.553} C_VEL
LIN {X 0,Y 347.846,Z 390.634,A -85,B 0,C 180,E1 -13652.745,E2 -13652.745} C_VEL
LIN {X 0,Y 347.782,Z 390.663,A -85,B 0,C 180,E1 -13656.162,E2 -13656.162} C_VEL
LIN {X 0,Y 347.806,Z 390.639,A -85,B 0,C 180,E1 -13659.91,E2 -13659.91} C_VEL
LIN {X 0,Y 347.86,Z 390.636,A -85,B 0,C 180,E1 -13662.36,E2 -13662.36} C_VEL
LIN {X 0,Y 347.891,Z 390.65,A -85,B 0,C 180,E1 -13665.971,E2 -13665.971} C_VEL
LIN {X 0,Y 347.925,Z 390.616,A -85,B 0,C 180,E1 -13669.526,E2 -13669.526} C_VEL
LIN {X 0,Y 348.068,Z 390.611,A -85,B 0,C 180,E1 -13671.875,E2 -13671.875} C_VEL
LIN {X 0,Y 348.062,Z 390.628,A -85,B 0,C 180,E1 -13674.206,E2 -13674.206} C_VEL
LIN {X 0,Y 348.203,Z 390.597,A -85,B 0,C 180,E1 -13677.687,E2 -13677.687} C_VEL
LIN {X 0,Y 348.321,Z 390.563,A -85,B 0,C 180,E1 -13680.001,E2 -13680.001} C_VEL
LIN {X 0,Y 348.203,Z 390.601,A -85,B 0,C 180,E1 -13682.314,E2 -13682.314} C_VEL
LIN {X 0,Y 348.102,Z 390.611,A -85,B 0,C 180,E1 -13686.958,E2 -13686.958} C_VEL
LIN {X 0,Y 347.923,Z 390.618,A -85,B 0,C 180,E1 -13690.475,E2 -13690.475} C_VEL
LIN {X 0,Y 347.894,Z 390.65,A -85,B 0,C 180,E1 -13694.151,E2 -13694.151} C_VEL
LIN {X 0,Y 347.886,Z 390.622,A -85,B 0,C 180,E1 -13698.291,E2 -13698.291} C_VEL
LIN {X 0,Y 347.785,Z 390.657,A -85,B 0,C 180,E1 -13701.636,E2 -13701.636} C_VEL
LIN {X 0,Y 347.809,Z 390.648,A -85,B 0,C 180,E1 -13705.109,E2 -13705.109} C_VEL
LIN {X 0,Y 347.809,Z 390.64,A -85,B 0,C 180,E1 -13707.695,E2 -13707.695} C_VEL
LIN {X 0,Y 347.768,Z 390.667,A -85,B 0,C 180,E1 -13710.347,E2 -13710.347} C_VEL
LIN {X 0,Y 347.746,Z 390.651,A -85,B 0,C 180,E1 -13714.045,E2 -13714.045} C_VEL
LIN {X 0,Y 347.765,Z 390.665,A -85,B 0,C 180,E1 -13717.321,E2 -13717.321} C_VEL
LIN {X 0,Y 347.792,Z 390.653,A -85,B 0,C 180,E1 -13720.289,E2 -13720.289} C_VEL
LIN {X 0,Y 347.814,Z 390.658,A -85,B 0,C 180,E1 -13723.395,E2 -13723.395} C_VEL
LIN {X 0,Y 347.728,Z 390.669,A -85,B 0,C 180,E1 -13726.687,E2 -13726.687} C_VEL
LIN {X 0,Y 347.746,Z 390.649,A -85,B 0,C 180,E1 -13730.174,E2 -13730.174} C_VEL
LIN {X 0,Y 347.762,Z 390.663,A -85,B 0,C 180,E1 -13732.68,E2 -13732.68} C_VEL
LIN {X 0,Y 347.749,Z 390.67,A -85,B 0,C 180,E1 -13735.957,E2 -13735.957} C_VEL
LIN {X 0,Y 347.821,Z 390.921,A -85,B 0,C 180,E1 -13737.703,E2 -13737.703} C_VEL
LIN {X 0,Y 349.463,Z 398.859,A -85,B 0,C 180,E1 -13740.565,E2 -13740.565} C_VEL
LIN {X 0,Y 350.958,Z 406.969,A -85,B 0,C 180,E1 -13743.221,E2 -13743.221} C_VEL
LIN {X 0,Y 351.012,Z 410.313,A -85,B 0,C 180,E1 -13744.29,E2 -13744.29} C_VEL
LIN {X 0,Y 349.979,Z 418.809,A -85,B 0,C 180,E1 -13746.915,E2 -13746.915} C_VEL
LIN {X 0,Y 350.766,Z 422.924,A -85,B 0,C 180,E1 -13747.121,E2 -13747.121} C_VEL
LIN {X 0,Y 355.516,Z 447.113,A -85,B 0,C 180,E1 -13747.957,E2 -13747.957} C_VEL
LIN {X 0,Y 356.908,Z 456.333,A -85,B 0,C 180,E1 -13748.242,E2 -13748.242} C_VEL
LIN {X 0,Y 355.667,Z 523.753,A -85,B 0,C 180,E1 -13749.619,E2 -13749.619} C_VEL
LIN {X 0,Y 355.229,Z 533.653,A -85,B 0,C 180,E1 -13749.933,E2 -13749.933} C_VEL
LIN {X 0,Y 354.582,Z 543.637,A -85,B 0,C 180,E1 -13750.385,E2 -13750.385} C_VEL
LIN {X 0,Y 353.733,Z 553.992,A -85,B 0,C 180,E1 -13751.014,E2 -13751.014} C_VEL
LIN {X 0,Y 352.906,Z 563.137,A -85,B 0,C 180,E1 -13751.721,E2 -13751.721} C_VEL
LIN {X 0,Y 351.936,Z 572.138,A -85,B 0,C 180,E1 -13752.57,E2 -13752.57} C_VEL
LIN {X 0,Y 350.976,Z 580.865,A -85,B 0,C 180,E1 -13753.571,E2 -13753.571} C_VEL
LIN {X 0,Y 350.042,Z 589.065,A -85,B 0,C 180,E1 -13754.698,E2 -13754.698} C_VEL
LIN {X 0,Y 349.096,Z 597.085,A -85,B 0,C 180,E1 -13756.02,E2 -13756.02} C_VEL
LIN {X 0,Y 348.367,Z 603.075,A -85,B 0,C 180,E1 -13757.179,E2 -13757.179} C_VEL
LIN {X 0,Y 347.561,Z 609.385,A -85,B 0,C 180,E1 -13758.63,E2 -13758.63} C_VEL
LIN {X 0,Y 347.03,Z 614.66,A -85,B 0,C 180,E1 -13760.088,E2 -13760.088} C_VEL
LIN {X 0,Y 346.556,Z 619.755,A -85,B 0,C 180,E1 -13761.839,E2 -13761.839} C_VEL
LIN {X 0,Y 346.345,Z 622.595,A -85,B 0,C 180,E1 -13763.007,E2 -13763.007} C_VEL
LIN {X 0,Y 346.164,Z 626.655,A -85,B 0,C 180,E1 -13765.342,E2 -13765.342} C_VEL
LIN {X 0,Y 346.143,Z 628.155,A -85,B 0,C 180,E1 -13766.508,E2 -13766.508} C_VEL
LIN {X 0,Y 346.104,Z 629.677,A -85,B 0,C 180,E1 -13768.837,E2 -13768.837} C_VEL
LIN {X 0,Y 346.148,Z 629.957,A -85,B 0,C 180,E1 -13770,E2 -13770} C_VEL
LIN {X 0,Y 346.084,Z 629.081,A -85,B 0,C 180,E1 -13772.328,E2 -13772.328} C_VEL
LIN {X 0,Y 346.143,Z 628.154,A -85,B 0,C 180,E1 -13773.492,E2 -13773.492} C_VEL
LIN {X 0,Y 346.2,Z 624.697,A -85,B 0,C 180,E1 -13775.885,E2 -13775.885} C_VEL
LIN {X 0,Y 346.467,Z 621.182,A -85,B 0,C 180,E1 -13777.577,E2 -13777.577} C_VEL
LIN {X 0,Y 346.862,Z 616.449,A -85,B 0,C 180,E1 -13779.329,E2 -13779.329} C_VEL
LIN {X 0,Y 347.462,Z 610.476,A -85,B 0,C 180,E1 -13781.079,E2 -13781.079} C_VEL
LIN {X 0,Y 347.997,Z 605.695,A -85,B 0,C 180,E1 -13782.243,E2 -13782.243} C_VEL
LIN {X 0,Y 348.736,Z 600.204,A -85,B 0,C 180,E1 -13783.401,E2 -13783.401} C_VEL
LIN {X 0,Y 349.73,Z 591.986,A -85,B 0,C 180,E1 -13784.846,E2 -13784.846} C_VEL
LIN {X 0,Y 350.663,Z 583.728,A -85,B 0,C 180,E1 -13786.055,E2 -13786.055} C_VEL
LIN {X 0,Y 351.526,Z 576.071,A -85,B 0,C 180,E1 -13787.002,E2 -13787.002} C_VEL
LIN {X 0,Y 352.576,Z 566.31,A -85,B 0,C 180,E1 -13787.997,E2 -13787.997} C_VEL
LIN {X 0,Y 353.429,Z 557.92,A -85,B 0,C 180,E1 -13788.702,E2 -13788.702} C_VEL
LIN {X 0,Y 354.261,Z 547.412,A -85,B 0,C 180,E1 -13789.408,E2 -13789.408} C_VEL
LIN {X 0,Y 355.062,Z 537.081,A -85,B 0,C 180,E1 -13789.927,E2 -13789.927} C_VEL
LIN {X 0,Y 355.611,Z 526.359,A -85,B 0,C 180,E1 -13790.31,E2 -13790.31} C_VEL
LIN {X 0,Y 356.058,Z 503.578,A -85,B 0,C 180,E1 -13790.811,E2 -13790.811} C_VEL
LIN {X 0,Y 356.887,Z 455.285,A -85,B 0,C 180,E1 -13791.781,E2 -13791.781} C_VEL
LIN {X 0,Y 352.192,Z 429.456,A -85,B 0,C 180,E1 -13792.641,E2 -13792.641} C_VEL
LIN {X 0,Y 349.955,Z 419.076,A -85,B 0,C 180,E1 -13793.051,E2 -13793.051} C_VEL
LIN {X 0,Y 350.021,Z 417.732,A -85,B 0,C 180,E1 -13793.363,E2 -13793.363} C_VEL
LIN {X 0,Y 351.12,Z 409.004,A -85,B 0,C 180,E1 -13796.126,E2 -13796.126} C_VEL
LIN {X 0,Y 350.319,Z 403.277,A -85,B 0,C 180,E1 -13798.027,E2 -13798.027} C_VEL
LIN {X 0,Y 348.399,Z 393.701,A -85,B 0,C 180,E1 -13801.294,E2 -13801.294} C_VEL
LIN {X 0,Y 347.797,Z 390.764,A -85,B 0,C 180,E1 -13802.376,E2 -13802.376} C_VEL
LIN {X 0,Y 347.773,Z 390.651,A -85,B 0,C 180,E1 -13806.065,E2 -13806.065} C_VEL
LIN {X 0,Y 347.755,Z 390.665,A -85,B 0,C 180,E1 -13808.792,E2 -13808.792} C_VEL
LIN {X 0,Y 347.753,Z 390.649,A -85,B 0,C 180,E1 -13811.83,E2 -13811.83} C_VEL
LIN {X 0,Y 347.799,Z 390.657,A -85,B 0,C 180,E1 -13815.011,E2 -13815.011} C_VEL
LIN {X 0,Y 347.788,Z 390.661,A -85,B 0,C 180,E1 -13818.39,E2 -13818.39} C_VEL
LIN {X 0,Y 347.78,Z 390.663,A -85,B 0,C 180,E1 -13822.01,E2 -13822.01} C_VEL
LIN {X 0,Y 347.746,Z 390.652,A -85,B 0,C 180,E1 -13825.536,E2 -13825.536} C_VEL
LIN {X 0,Y 347.765,Z 390.666,A -85,B 0,C 180,E1 -13828.302,E2 -13828.302} C_VEL
LIN {X 0,Y 347.807,Z 390.655,A -85,B 0,C 180,E1 -13830.99,E2 -13830.99} C_VEL
LIN {X 0,Y 347.832,Z 390.634,A -85,B 0,C 180,E1 -13833.607,E2 -13833.607} C_VEL
LIN {X 0,Y 347.789,Z 390.662,A -85,B 0,C 180,E1 -13836.161,E2 -13836.161} C_VEL
LIN {X 0,Y 347.812,Z 390.641,A -85,B 0,C 180,E1 -13839.909,E2 -13839.909} C_VEL
LIN {X 0,Y 347.866,Z 390.629,A -85,B 0,C 180,E1 -13842.359,E2 -13842.359} C_VEL
LIN {X 0,Y 347.897,Z 390.648,A -85,B 0,C 180,E1 -13845.97,E2 -13845.97} C_VEL
LIN {X 0,Y 347.927,Z 390.617,A -85,B 0,C 180,E1 -13849.525,E2 -13849.525} C_VEL
LIN {X 0,Y 348.106,Z 390.611,A -85,B 0,C 180,E1 -13853.042,E2 -13853.042} C_VEL
LIN {X 0,Y 348.206,Z 390.6,A -85,B 0,C 180,E1 -13857.686,E2 -13857.686} C_VEL
LIN {X 0,Y 348.323,Z 390.563,A -85,B 0,C 180,E1 -13859.999,E2 -13859.999} C_VEL
LIN {X 0,Y 348.207,Z 390.596,A -85,B 0,C 180,E1 -13862.313,E2 -13862.313} C_VEL
LIN {X 0,Y 348.104,Z 390.62,A -85,B 0,C 180,E1 -13866.957,E2 -13866.957} C_VEL
LIN {X 0,Y 347.966,Z 390.613,A -85,B 0,C 180,E1 -13869.298,E2 -13869.298} C_VEL
LIN {X 0,Y 347.891,Z 390.641,A -85,B 0,C 180,E1 -13872.839,E2 -13872.839} C_VEL
LIN {X 0,Y 347.837,Z 390.65,A -85,B 0,C 180,E1 -13876.431,E2 -13876.431} C_VEL
LIN {X 0,Y 347.848,Z 390.629,A -85,B 0,C 180,E1 -13878.86,E2 -13878.86} C_VEL
LIN {X 0,Y 347.771,Z 390.662,A -85,B 0,C 180,E1 -13882.579,E2 -13882.579} C_VEL
LIN {X 0,Y 347.809,Z 390.656,A -85,B 0,C 180,E1 -13885.108,E2 -13885.108} C_VEL
LIN {X 0,Y 347.805,Z 390.64,A -85,B 0,C 180,E1 -13887.694,E2 -13887.694} C_VEL
LIN {X 0,Y 347.746,Z 390.666,A -85,B 0,C 180,E1 -13890.347,E2 -13890.347} C_VEL
LIN {X 0,Y 347.745,Z 390.65,A -85,B 0,C 180,E1 -13894.043,E2 -13894.043} C_VEL
LIN {X 0,Y 347.762,Z 390.668,A -85,B 0,C 180,E1 -13897.32,E2 -13897.32} C_VEL
LIN {X 0,Y 347.728,Z 390.657,A -85,B 0,C 180,E1 -13900.297,E2 -13900.297} C_VEL
LIN {X 0,Y 347.724,Z 390.673,A -85,B 0,C 180,E1 -13903.407,E2 -13903.407} C_VEL
LIN {X 0,Y 347.722,Z 390.637,A -85,B 0,C 180,E1 -13906.686,E2 -13906.686} C_VEL
LIN {X 0,Y 347.753,Z 390.65,A -85,B 0,C 180,E1 -13910.171,E2 -13910.171} C_VEL
LIN {X 0,Y 347.765,Z 390.667,A -85,B 0,C 180,E1 -13912.68,E2 -13912.68} C_VEL
LIN {X 0,Y 347.744,Z 390.643,A -85,B 0,C 180,E1 -13915.956,E2 -13915.956} C_VEL
LIN {X 0,Y 347.761,Z 390.654,A -85,B 0,C 180,E1 -13919.653,E2 -13919.653} C_VEL
LIN {X 0,Y 347.849,Z 390.657,A -85,B 0,C 180,E1 -13922.744,E2 -13922.744} C_VEL
LIN {X 0,Y 347.785,Z 390.666,A -85,B 0,C 180,E1 -13926.162,E2 -13926.162} C_VEL
LIN {X 0,Y 347.822,Z 390.782,A -85,B 0,C 180,E1 -13929.137,E2 -13929.137} C_VEL
LIN {X 0,Y 348.019,Z 391.795,A -85,B 0,C 180,E1 -13929.459,E2 -13929.459} C_VEL
LIN {X 0,Y 349.598,Z 394.589,A -85,B 0,C 180,E1 -13929.907,E2 -13929.907} C_VEL
LIN {X 0,Y 351.802,Z 396.47,A -85,B 0,C 180,E1 -13930.408,E2 -13930.408} C_VEL
LIN {X 0,Y 353.932,Z 399.738,A -85,B 0,C 180,E1 -13930.994,E2 -13930.994} C_VEL
LIN {X 0,Y 356.629,Z 402.243,A -85,B 0,C 180,E1 -13931.667,E2 -13931.667} C_VEL
LIN {X 0,Y 358.936,Z 405.379,A -85,B 0,C 180,E1 -13932.324,E2 -13932.324} C_VEL
LIN {X 0,Y 361.878,Z 408.01,A -85,B 0,C 180,E1 -13933.126,E2 -13933.126} C_VEL
LIN {X 0,Y 364.508,Z 411.265,A -85,B 0,C 180,E1 -13933.937,E2 -13933.937} C_VEL
LIN {X 0,Y 367.946,Z 414.098,A -85,B 0,C 180,E1 -13934.973,E2 -13934.973} C_VEL
LIN {X 0,Y 370.997,Z 417.698,A -85,B 0,C 180,E1 -13936.035,E2 -13936.035} C_VEL
LIN {X 0,Y 374.481,Z 420.472,A -85,B 0,C 180,E1 -13937.295,E2 -13937.295} C_VEL
LIN {X 0,Y 377.297,Z 423.682,A -85,B 0,C 180,E1 -13938.458,E2 -13938.458} C_VEL
LIN {X 0,Y 380.314,Z 426.016,A -85,B 0,C 180,E1 -13939.787,E2 -13939.787} C_VEL
LIN {X 0,Y 382.292,Z 427.049,A -85,B 0,C 180,E1 -13940.718,E2 -13940.718} C_VEL
LIN {X 0,Y 385.025,Z 430.424,A -85,B 0,C 180,E1 -13942.364,E2 -13942.364} C_VEL
LIN {X 0,Y 387.586,Z 432.48,A -85,B 0,C 180,E1 -13944.253,E2 -13944.253} C_VEL
LIN {X 0,Y 389.26,Z 433.367,A -85,B 0,C 180,E1 -13945.858,E2 -13945.858} C_VEL
LIN {X 0,Y 390.395,Z 433.748,A -85,B 0,C 180,E1 -13947.439,E2 -13947.439} C_VEL
LIN {X 0,Y 390.961,Z 434.179,A -85,B 0,C 180,E1 -13948.97,E2 -13948.97} C_VEL
LIN {X 0,Y 391.134,Z 434.117,A -85,B 0,C 180,E1 -13950,E2 -13950} C_VEL
LIN {X 0,Y 390.864,Z 434.04,A -85,B 0,C 180,E1 -13951.545,E2 -13951.545} C_VEL
LIN {X 0,Y 390.115,Z 433.611,A -85,B 0,C 180,E1 -13953.098,E2 -13953.098} C_VEL
LIN {X 0,Y 388.502,Z 433.035,A -85,B 0,C 180,E1 -13954.929,E2 -13954.929} C_VEL
LIN {X 0,Y 386.388,Z 431.598,A -85,B 0,C 180,E1 -13956.669,E2 -13956.669} C_VEL
LIN {X 0,Y 384.295,Z 429.694,A -85,B 0,C 180,E1 -13958.071,E2 -13958.071} C_VEL
LIN {X 0,Y 382.055,Z 426.876,A -85,B 0,C 180,E1 -13959.396,E2 -13959.396} C_VEL
LIN {X 0,Y 378.835,Z 424.995,A -85,B 0,C 180,E1 -13960.894,E2 -13960.894} C_VEL
LIN {X 0,Y 375.554,Z 421.771,A -85,B 0,C 180,E1 -13962.29,E2 -13962.29} C_VEL
LIN {X 0,Y 373.78,Z 419.8,A -85,B 0,C 180,E1 -13962.97,E2 -13962.97} C_VEL
LIN {X 0,Y 370.641,Z 417.366,A -85,B 0,C 180,E1 -13964.084,E2 -13964.084} C_VEL
LIN {X 0,Y 367.767,Z 413.857,A -85,B 0,C 180,E1 -13965.087,E2 -13965.087} C_VEL
LIN {X 0,Y 363.716,Z 410.414,A -85,B 0,C 180,E1 -13966.311,E2 -13966.311} C_VEL
LIN {X 0,Y 360.955,Z 407.107,A -85,B 0,C 180,E1 -13967.125,E2 -13967.125} C_VEL
LIN {X 0,Y 358.033,Z 404.343,A -85,B 0,C 180,E1 -13967.937,E2 -13967.937} C_VEL
LIN {X 0,Y 356.111,Z 401.532,A -85,B 0,C 180,E1 -13968.468,E2 -13968.468} C_VEL
LIN {X 0,Y 353.384,Z 399.096,A -85,B 0,C 180,E1 -13969.15,E2 -13969.15} C_VEL
LIN {X 0,Y 351.549,Z 396.079,A -85,B 0,C 180,E1 -13969.658,E2 -13969.658} C_VEL
LIN {X 0,Y 349.139,Z 394.032,A -85,B 0,C 180,E1 -13970.203,E2 -13970.203} C_VEL
LIN {X 0,Y 347.916,Z 391.339,A -85,B 0,C 180,E1 -13970.624,E2 -13970.624} C_VEL
LIN {X 0,Y 347.81,Z 390.699,A -85,B 0,C 180,E1 -13971.017,E2 -13971.017} C_VEL
LIN {X 0,Y 347.807,Z 390.662,A -85,B 0,C 180,E1 -13975.108,E2 -13975.108} C_VEL
LIN {X 0,Y 347.807,Z 390.658,A -85,B 0,C 180,E1 -13977.693,E2 -13977.693} C_VEL
LIN {X 0,Y 347.759,Z 390.654,A -85,B 0,C 180,E1 -13980.346,E2 -13980.346} C_VEL
LIN {X 0,Y 347.738,Z 390.642,A -85,B 0,C 180,E1 -13984.464,E2 -13984.464} C_VEL
LIN {X 0,Y 347.775,Z 390.665,A -85,B 0,C 180,E1 -13987.99,E2 -13987.99} C_VEL
LIN {X 0,Y 347.752,Z 390.622,A -85,B 0,C 180,E1 -13991.829,E2 -13991.829} C_VEL
LIN {X 0,Y 347.76,Z 390.658,A -85,B 0,C 180,E1 -13995.017,E2 -13995.017} C_VEL
LIN {X 0,Y 347.761,Z 390.657,A -85,B 0,C 180,E1 -13998.394,E2 -13998.394} C_VEL
LIN {X 0,Y 347.772,Z 390.665,A -85,B 0,C 180,E1 -14002.01,E2 -14002.01} C_VEL
LIN {X 0,Y 347.737,Z 390.65,A -85,B 0,C 180,E1 -14005.536,E2 -14005.536} C_VEL
LIN {X 0,Y 347.75,Z 390.665,A -85,B 0,C 180,E1 -14009.553,E2 -14009.553} C_VEL
LIN {X 0,Y 347.143,Z 390.743,A -85,B 0,C 180,E1 -14010.521,E2 -14010.521} C_VEL
LIN {X 0,Y 344.319,Z 391.087,A -85,B 0,C 180,E1 -14012.096,E2 -14012.096} C_VEL
LIN {X 0,Y 341.89,Z 391.384,A -85,B 0,C 180,E1 -14013.37,E2 -14013.37} C_VEL
LIN {X 0,Y 340.841,Z 391.516,A -85,B 0,C 180,E1 -14014.357,E2 -14014.357} C_VEL
LIN {X 0,Y 340.755,Z 391.53,A -85,B 0,C 180,E1 -14014.691,E2 -14014.691} C_VEL
LIN {X 0,Y 340.735,Z 391.536,A -85,B 0,C 180,E1 -14018.207,E2 -14018.207} C_VEL
LIN {X 0,Y 340.851,Z 391.505,A -85,B 0,C 180,E1 -14021.985,E2 -14021.985} C_VEL
LIN {X 0,Y 340.863,Z 391.524,A -85,B 0,C 180,E1 -14025.705,E2 -14025.705} C_VEL
LIN {X 0,Y 340.868,Z 391.495,A -85,B 0,C 180,E1 -14029.307,E2 -14029.307} C_VEL
LIN {X 0,Y 341.069,Z 391.496,A -85,B 0,C 180,E1 -14032.899,E2 -14032.899} C_VEL
LIN {X 0,Y 341.165,Z 391.473,A -85,B 0,C 180,E1 -14037.639,E2 -14037.639} C_VEL
LIN {X 0,Y 341.272,Z 391.441,A -85,B 0,C 180,E1 -14040.001,E2 -14040.001} C_VEL
LIN {X 0,Y 341.165,Z 391.478,A -85,B 0,C 180,E1 -14042.362,E2 -14042.362} C_VEL
LIN {X 0,Y 341.072,Z 391.486,A -85,B 0,C 180,E1 -14047.103,E2 -14047.103} C_VEL
LIN {X 0,Y 340.866,Z 391.5,A -85,B 0,C 180,E1 -14050.695,E2 -14050.695} C_VEL
LIN {X 0,Y 340.859,Z 391.525,A -85,B 0,C 180,E1 -14054.326,E2 -14054.326} C_VEL
LIN {X 0,Y 340.833,Z 391.5,A -85,B 0,C 180,E1 -14058.467,E2 -14058.467} C_VEL
LIN {X 0,Y 340.75,Z 391.535,A -85,B 0,C 180,E1 -14061.858,E2 -14061.858} C_VEL
LIN {X 0,Y 340.769,Z 391.519,A -85,B 0,C 180,E1 -14065.665,E2 -14065.665} C_VEL
LIN {X 0,Y 340.739,Z 391.527,A -85,B 0,C 180,E1 -14068.32,E2 -14068.32} C_VEL
LIN {X 0,Y 340.713,Z 391.542,A -85,B 0,C 180,E1 -14071.044,E2 -14071.044} C_VEL
LIN {X 0,Y 340.717,Z 391.534,A -85,B 0,C 180,E1 -14075.28,E2 -14075.28} C_VEL
LIN {X 0,Y 340.718,Z 391.538,A -85,B 0,C 180,E1 -14078.389,E2 -14078.389} C_VEL
LIN {X 0,Y 340.726,Z 391.539,A -85,B 0,C 180,E1 -14081.304,E2 -14081.304} C_VEL
LIN {X 0,Y 340.743,Z 391.534,A -85,B 0,C 180,E1 -14084.53,E2 -14084.53} C_VEL
LIN {X 0,Y 340.685,Z 391.525,A -85,B 0,C 180,E1 -14088.691,E2 -14088.691} C_VEL
LIN {X 0,Y 340.733,Z 391.543,A -85,B 0,C 180,E1 -14091.774,E2 -14091.774} C_VEL
LIN {X 0,Y 340.723,Z 391.543,A -85,B 0,C 180,E1 -14095.596,E2 -14095.596} C_VEL
LIN {X 0,Y 340.758,Z 391.781,A -85,B 0,C 180,E1 -14097.31,E2 -14097.31} C_VEL
LIN {X 0,Y 342.353,Z 399.242,A -85,B 0,C 180,E1 -14100.077,E2 -14100.077} C_VEL
LIN {X 0,Y 343.92,Z 407.813,A -85,B 0,C 180,E1 -14102.957,E2 -14102.957} C_VEL
LIN {X 0,Y 344.109,Z 410.856,A -85,B 0,C 180,E1 -14103.982,E2 -14103.982} C_VEL
LIN {X 0,Y 343.135,Z 418.525,A -85,B 0,C 180,E1 -14106.41,E2 -14106.41} C_VEL
LIN {X 0,Y 343.424,Z 420.542,A -85,B 0,C 180,E1 -14106.554,E2 -14106.554} C_VEL
LIN {X 0,Y 348.76,Z 447.046,A -85,B 0,C 180,E1 -14107.51,E2 -14107.51} C_VEL
LIN {X 0,Y 350.322,Z 457.187,A -85,B 0,C 180,E1 -14107.834,E2 -14107.834} C_VEL
LIN {X 0,Y 349.029,Z 523.565,A -85,B 0,C 180,E1 -14109.214,E2 -14109.214} C_VEL
LIN {X 0,Y 348.581,Z 533.458,A -85,B 0,C 180,E1 -14109.533,E2 -14109.533} C_VEL
LIN {X 0,Y 347.912,Z 543.443,A -85,B 0,C 180,E1 -14109.993,E2 -14109.993} C_VEL
LIN {X 0,Y 347.025,Z 553.797,A -85,B 0,C 180,E1 -14110.633,E2 -14110.633} C_VEL
LIN {X 0,Y 346.169,Z 562.942,A -85,B 0,C 180,E1 -14111.352,E2 -14111.352} C_VEL
LIN {X 0,Y 345.144,Z 571.942,A -85,B 0,C 180,E1 -14112.216,E2 -14112.216} C_VEL
LIN {X 0,Y 344.135,Z 580.669,A -85,B 0,C 180,E1 -14113.235,E2 -14113.235} C_VEL
LIN {X 0,Y 343.137,Z 588.869,A -85,B 0,C 180,E1 -14114.382,E2 -14114.382} C_VEL
LIN {X 0,Y 342.165,Z 596.889,A -85,B 0,C 180,E1 -14115.731,E2 -14115.731} C_VEL
LIN {X 0,Y 341.421,Z 602.88,A -85,B 0,C 180,E1 -14116.914,E2 -14116.914} C_VEL
LIN {X 0,Y 340.566,Z 609.189,A -85,B 0,C 180,E1 -14118.393,E2 -14118.393} C_VEL
LIN {X 0,Y 340.026,Z 614.465,A -85,B 0,C 180,E1 -14119.882,E2 -14119.882} C_VEL
LIN {X 0,Y 339.515,Z 619.559,A -85,B 0,C 180,E1 -14121.669,E2 -14121.669} C_VEL
LIN {X 0,Y 339.2,Z 623.524,A -85,B 0,C 180,E1 -14123.457,E2 -14123.457} C_VEL
LIN {X 0,Y 339.071,Z 626.459,A -85,B 0,C 180,E1 -14125.245,E2 -14125.245} C_VEL
LIN {X 0,Y 339.067,Z 627.96,A -85,B 0,C 180,E1 -14126.435,E2 -14126.435} C_VEL
LIN {X 0,Y 339.007,Z 629.482,A -85,B 0,C 180,E1 -14128.812,E2 -14128.812} C_VEL
LIN {X 0,Y 339.051,Z 629.762,A -85,B 0,C 180,E1 -14130,E2 -14130} C_VEL
LIN {X 0,Y 338.999,Z 628.886,A -85,B 0,C 180,E1 -14132.377,E2 -14132.377} C_VEL
LIN {X 0,Y 339.067,Z 627.96,A -85,B 0,C 180,E1 -14133.565,E2 -14133.565} C_VEL
LIN {X 0,Y 339.115,Z 624.611,A -85,B 0,C 180,E1 -14135.948,E2 -14135.948} C_VEL
LIN {X 0,Y 339.398,Z 620.986,A -85,B 0,C 180,E1 -14137.736,E2 -14137.736} C_VEL
LIN {X 0,Y 339.817,Z 616.253,A -85,B 0,C 180,E1 -14139.524,E2 -14139.524} C_VEL
LIN {X 0,Y 340.457,Z 610.28,A -85,B 0,C 180,E1 -14141.31,E2 -14141.31} C_VEL
LIN {X 0,Y 341.047,Z 605.499,A -85,B 0,C 180,E1 -14142.496,E2 -14142.496} C_VEL
LIN {X 0,Y 341.815,Z 600.008,A -85,B 0,C 180,E1 -14143.677,E2 -14143.677} C_VEL
LIN {X 0,Y 342.864,Z 591.79,A -85,B 0,C 180,E1 -14145.15,E2 -14145.15} C_VEL
LIN {X 0,Y 343.778,Z 583.748,A -85,B 0,C 180,E1 -14146.355,E2 -14146.355} C_VEL
LIN {X 0,Y 344.74,Z 575.876,A -85,B 0,C 180,E1 -14147.347,E2 -14147.347} C_VEL
LIN {X 0,Y 345.826,Z 566.114,A -85,B 0,C 180,E1 -14148.361,E2 -14148.361} C_VEL
LIN {X 0,Y 346.701,Z 557.725,A -85,B 0,C 180,E1 -14149.079,E2 -14149.079} C_VEL
LIN {X 0,Y 347.562,Z 547.216,A -85,B 0,C 180,E1 -14149.798,E2 -14149.798} C_VEL
LIN {X 0,Y 348.381,Z 536.885,A -85,B 0,C 180,E1 -14150.326,E2 -14150.326} C_VEL
LIN {X 0,Y 348.972,Z 526.164,A -85,B 0,C 180,E1 -14150.714,E2 -14150.714} C_VEL
LIN {X 0,Y 349.432,Z 503.383,A -85,B 0,C 180,E1 -14151.225,E2 -14151.225} C_VEL
LIN {X 0,Y 350.303,Z 456.378,A -85,B 0,C 180,E1 -14152.185,E2 -14152.185} C_VEL
LIN {X 0,Y 345.812,Z 431.486,A -85,B 0,C 180,E1 -14153.034,E2 -14153.034} C_VEL
LIN {X 0,Y 343.106,Z 418.809,A -85,B 0,C 180,E1 -14153.545,E2 -14153.545} C_VEL
LIN {X 0,Y 343.328,Z 416.589,A -85,B 0,C 180,E1 -14154.167,E2 -14154.167} C_VEL
LIN {X 0,Y 344.161,Z 410.082,A -85,B 0,C 180,E1 -14156.271,E2 -14156.271} C_VEL
LIN {X 0,Y 343.026,Z 402.662,A -85,B 0,C 180,E1 -14158.814,E2 -14158.814} C_VEL
LIN {X 0,Y 340.973,Z 392.736,A -85,B 0,C 180,E1 -14162.319,E2 -14162.319} C_VEL
LIN {X 0,Y 340.735,Z 391.637,A -85,B 0,C 180,E1 -14162.781,E2 -14162.781} C_VEL
LIN {X 0,Y 340.713,Z 391.531,A -85,B 0,C 180,E1 -14166.44,E2 -14166.44} C_VEL
LIN {X 0,Y 340.701,Z 391.526,A -85,B 0,C 180,E1 -14169.752,E2 -14169.752} C_VEL
LIN {X 0,Y 340.68,Z 391.546,A -85,B 0,C 180,E1 -14172.903,E2 -14172.903} C_VEL
LIN {X 0,Y 340.756,Z 391.533,A -85,B 0,C 180,E1 -14176.208,E2 -14176.208} C_VEL
LIN {X 0,Y 340.766,Z 391.528,A -85,B 0,C 180,E1 -14179.737,E2 -14179.737} C_VEL
LIN {X 0,Y 340.713,Z 391.545,A -85,B 0,C 180,E1 -14183.558,E2 -14183.558} C_VEL
LIN {X 0,Y 340.696,Z 391.528,A -85,B 0,C 180,E1 -14186.153,E2 -14186.153} C_VEL
LIN {X 0,Y 340.776,Z 391.533,A -85,B 0,C 180,E1 -14190.332,E2 -14190.332} C_VEL
LIN {X 0,Y 340.806,Z 391.508,A -85,B 0,C 180,E1 -14193.019,E2 -14193.019} C_VEL
LIN {X 0,Y 340.729,Z 391.538,A -85,B 0,C 180,E1 -14196.927,E2 -14196.927} C_VEL
LIN {X 0,Y 340.79,Z 391.509,A -85,B 0,C 180,E1 -14200.733,E2 -14200.733} C_VEL
LIN {X 0,Y 340.787,Z 391.516,A -85,B 0,C 180,E1 -14203.218,E2 -14203.218} C_VEL
LIN {X 0,Y 340.843,Z 391.523,A -85,B 0,C 180,E1 -14206.89,E2 -14206.89} C_VEL
LIN {X 0,Y 340.928,Z 391.479,A -85,B 0,C 180,E1 -14210.507,E2 -14210.507} C_VEL
LIN {X 0,Y 341.076,Z 391.486,A -85,B 0,C 180,E1 -14212.898,E2 -14212.898} C_VEL
LIN {X 0,Y 341.168,Z 391.477,A -85,B 0,C 180,E1 -14217.638,E2 -14217.638} C_VEL
LIN {X 0,Y 341.274,Z 391.44,A -85,B 0,C 180,E1 -14219.999,E2 -14219.999} C_VEL
LIN {X 0,Y 341.168,Z 391.473,A -85,B 0,C 180,E1 -14222.361,E2 -14222.361} C_VEL
LIN {X 0,Y 341.073,Z 391.495,A -85,B 0,C 180,E1 -14227.101,E2 -14227.101} C_VEL
LIN {X 0,Y 340.871,Z 391.495,A -85,B 0,C 180,E1 -14230.693,E2 -14230.693} C_VEL
LIN {X 0,Y 340.861,Z 391.524,A -85,B 0,C 180,E1 -14234.324,E2 -14234.324} C_VEL
LIN {X 0,Y 340.834,Z 391.505,A -85,B 0,C 180,E1 -14238.466,E2 -14238.466} C_VEL
LIN {X 0,Y 340.751,Z 391.535,A -85,B 0,C 180,E1 -14241.856,E2 -14241.856} C_VEL
LIN {X 0,Y 340.769,Z 391.525,A -85,B 0,C 180,E1 -14245.664,E2 -14245.664} C_VEL
LIN {X 0,Y 340.725,Z 391.526,A -85,B 0,C 180,E1 -14248.32,E2 -14248.32} C_VEL
LIN {X 0,Y 340.694,Z 391.547,A -85,B 0,C 180,E1 -14251.044,E2 -14251.044} C_VEL
LIN {X 0,Y 340.715,Z 391.527,A -85,B 0,C 180,E1 -14255.278,E2 -14255.278} C_VEL
LIN {X 0,Y 340.708,Z 391.544,A -85,B 0,C 180,E1 -14258.386,E2 -14258.386} C_VEL
LIN {X 0,Y 340.696,Z 391.543,A -85,B 0,C 180,E1 -14262.045,E2 -14262.045} C_VEL
LIN {X 0,Y 340.679,Z 391.533,A -85,B 0,C 180,E1 -14265.461,E2 -14265.461} C_VEL
LIN {X 0,Y 340.695,Z 391.503,A -85,B 0,C 180,E1 -14268.692,E2 -14268.692} C_VEL
LIN {X 0,Y 340.742,Z 391.543,A -85,B 0,C 180,E1 -14271.774,E2 -14271.774} C_VEL
LIN {X 0,Y 340.719,Z 391.515,A -85,B 0,C 180,E1 -14275.595,E2 -14275.595} C_VEL
LIN {X 0,Y 340.701,Z 391.542,A -85,B 0,C 180,E1 -14278.956,E2 -14278.956} C_VEL
LIN {X 0,Y 340.776,Z 391.536,A -85,B 0,C 180,E1 -14282.473,E2 -14282.473} C_VEL
LIN {X 0,Y 340.752,Z 391.541,A -85,B 0,C 180,E1 -14285.638,E2 -14285.638} C_VEL
LIN {X 0,Y 340.749,Z 391.652,A -85,B 0,C 180,E1 -14287.813,E2 -14287.813} C_VEL
LIN {X 0,Y 340.931,Z 392.489,A -85,B 0,C 180,E1 -14288.111,E2 -14288.111} C_VEL
LIN {X 0,Y 342.359,Z 395.226,A -85,B 0,C 180,E1 -14288.51,E2 -14288.51} C_VEL
LIN {X 0,Y 344.49,Z 397.308,A -85,B 0,C 180,E1 -14288.961,E2 -14288.961} C_VEL
LIN {X 0,Y 346.856,Z 400.754,A -85,B 0,C 180,E1 -14289.549,E2 -14289.549} C_VEL
LIN {X 0,Y 348.969,Z 402.833,A -85,B 0,C 180,E1 -14290.042,E2 -14290.042} C_VEL
LIN {X 0,Y 351.718,Z 406.35,A -85,B 0,C 180,E1 -14290.721,E2 -14290.721} C_VEL
LIN {X 0,Y 353.899,Z 408.475,A -85,B 0,C 180,E1 -14291.279,E2 -14291.279} C_VEL
LIN {X 0,Y 357.055,Z 412.207,A -85,B 0,C 180,E1 -14292.106,E2 -14292.106} C_VEL
LIN {X 0,Y 359.357,Z 414.244,A -85,B 0,C 180,E1 -14292.742,E2 -14292.742} C_VEL
LIN {X 0,Y 362.473,Z 417.787,A -85,B 0,C 180,E1 -14293.634,E2 -14293.634} C_VEL
LIN {X 0,Y 365.929,Z 420.725,A -85,B 0,C 180,E1 -14294.673,E2 -14294.673} C_VEL
LIN {X 0,Y 369.17,Z 424.335,A -85,B 0,C 180,E1 -14295.766,E2 -14295.766} C_VEL
LIN {X 0,Y 372.814,Z 427.223,A -85,B 0,C 180,E1 -14297.04,E2 -14297.04} C_VEL
LIN {X 0,Y 376.091,Z 430.742,A -85,B 0,C 180,E1 -14298.35,E2 -14298.35} C_VEL
LIN {X 0,Y 379.346,Z 433.075,A -85,B 0,C 180,E1 -14299.761,E2 -14299.761} C_VEL
LIN {X 0,Y 381.145,Z 434.141,A -85,B 0,C 180,E1 -14300.617,E2 -14300.617} C_VEL
